	//Alarm Priority setpoint
	{attribute 'OPC.UA.DA' :='1'}
	popa_0081_lt_3202_a_high_high_priority : INT;
	//Alarm delay setpoint(seconds)
	{attribute 'OPC.UA.DA' :='1'}
	popa_0081_lt_3202_a_high_high_delay_setpoint : INT;
	//Alarm active for HMI
	{attribute 'OPC.UA.DA' :='1'}
	popa_0081_lt_3202_a_high_high_active : BOOL;
	//Analog Alarm Setpoint
	{attribute 'OPC.UA.DA' :='1'}
	popa_0081_lt_3202_a_high_high_setpoint : REAL;
	//Alarm enable
	{attribute 'OPC.UA.DA' :='1'}
	popa_0081_lt_3202_a_high_high_enable: BOOL;
	
	
	//Raw Min value for analog input
	{attribute 'OPC.UA.DA' :='1'}
	popa_0081_lt_3202_a_raw_min : REAL :=0;
	//Raw max value for analog input
	{attribute 'OPC.UA.DA' :='1'}
	popa_0081_lt_3202_a_raw_max : REAL :=32767;
	//EU Min value for analog input
	{attribute 'OPC.UA.DA' :='1'}
	popa_0081_lt_3202_a_eu_min : REAL;
	//EU Max value for analog input
	{attribute 'OPC.UA.DA' :='1'}
	popa_0081_lt_3202_a_eu_max : REAL;
	//Filter factor value for analog input
	{attribute 'OPC.UA.DA' :='1'}
	popa_0081_lt_3202_a_filter_factor : REAL;
	//Scaled value for analog input
	{attribute 'OPC.UA.DA' :='1'}
	popa_0081_lt_3202_a_scaled_value : REAL;
	
	//---lt_3302-----------------------------------------------------------------------------------------------------------------------
	//Alarm Priority setpoint
	{attribute 'OPC.UA.DA' :='1'}
	popa_0081_lt_3302_a_low_low_priority : INT;
	//Alarm delay setpoint(seconds)
	{attribute 'OPC.UA.DA' :='1'}
	popa_0081_lt_3302_a_low_low_delay_setpoint : INT;
	//Alarm active for HMI
	{attribute 'OPC.UA.DA' :='1'}
	popa_0081_lt_3302_a_low_low_active : BOOL;
	//Analog Alarm Setpoint
	{attribute 'OPC.UA.DA' :='1'}
	popa_0081_lt_3302_a_low_low_setpoint : REAL;
	//Alarm enable
	{attribute 'OPC.UA.DA' :='1'}
	popa_0081_lt_3302_a_low_low_enable: BOOL;
	
	//Alarm Priority setpoint
	{attribute 'OPC.UA.DA' :='1'}
	popa_0081_lt_3302_a_low_priority : INT;
	//Alarm delay setpoint(seconds)
	{attribute 'OPC.UA.DA' :='1'}
	popa_0081_lt_3302_a_low_delay_setpoint : INT;
	//Alarm active for HMI
	{attribute 'OPC.UA.DA' :='1'}
	popa_0081_lt_3302_a_low_active : BOOL;
	//Analog Alarm Setpoint
	{attribute 'OPC.UA.DA' :='1'}
	popa_0081_lt_3302_a_low_setpoint : REAL;
	//Alarm enable
	{attribute 'OPC.UA.DA' :='1'}
	popa_0081_lt_3302_a_low_enable: BOOL;
	
	//Alarm Priority setpoint
	{attribute 'OPC.UA.DA' :='1'}
	popa_0081_lt_3302_a_high_priority : INT;
	//Alarm delay setpoint(seconds)
	{attribute 'OPC.UA.DA' :='1'}
	popa_0081_lt_3302_a_high_delay_setpoint : INT;
	//Alarm active for HMI
	{attribute 'OPC.UA.DA' :='1'}
	popa_0081_lt_3302_a_high_active : BOOL;
	//Analog Alarm Setpoint
	{attribute 'OPC.UA.DA' :='1'}
	popa_0081_lt_3302_a_high_setpoint : REAL;
	//Alarm enable
	{attribute 'OPC.UA.DA' :='1'}
	popa_0081_lt_3302_a_high_enable: BOOL;
	
	//Alarm Priority setpoint
	{attribute 'OPC.UA.DA' :='1'}
	popa_0081_lt_3302_a_high_high_priority : INT;
	//Alarm delay setpoint(seconds)
	{attribute 'OPC.UA.DA' :='1'}
	popa_0081_lt_3302_a_high_high_delay_setpoint : INT;
	//Alarm active for HMI
	{attribute 'OPC.UA.DA' :='1'}
	popa_0081_lt_3302_a_high_high_active : BOOL;
	//Analog Alarm Setpoint
	{attribute 'OPC.UA.DA' :='1'}
	popa_0081_lt_3302_a_high_high_setpoint : REAL;
	//Alarm enable
	{attribute 'OPC.UA.DA' :='1'}
	popa_0081_lt_3302_a_high_high_enable: BOOL;
	
	
	//Raw Min value for analog input
	{attribute 'OPC.UA.DA' :='1'}
	popa_0081_lt_3302_a_raw_min : REAL :=0;
	//Raw max value for analog input
	{attribute 'OPC.UA.DA' :='1'}
	popa_0081_lt_3302_a_raw_max : REAL :=32767;
	//EU Min value for analog input
	{attribute 'OPC.UA.DA' :='1'}
	popa_0081_lt_3302_a_eu_min : REAL;
	//EU Max value for analog input
	{attribute 'OPC.UA.DA' :='1'}
	popa_0081_lt_3302_a_eu_max : REAL;
	//Filter factor value for analog input
	{attribute 'OPC.UA.DA' :='1'}
	popa_0081_lt_3302_a_filter_factor : REAL;
	//Scaled value for analog input
	{attribute 'OPC.UA.DA' :='1'}
	popa_0081_lt_3302_a_scaled_value : REAL;
	
	//---lt_3153-----------------------------------------------------------------------------------------------------------------------
	//Alarm Priority setpoint
	{attribute 'OPC.UA.DA' :='1'}
	popa_0081_lt_3153_a_low_low_priority : INT;
	//Alarm delay setpoint(seconds)
	{attribute 'OPC.UA.DA' :='1'}
	popa_0081_lt_3153_a_low_low_delay_setpoint : INT;
	//Alarm active for HMI
	{attribute 'OPC.UA.DA' :='1'}
	popa_0081_lt_3153_a_low_low_active : BOOL;
	//Analog Alarm Setpoint
	{attribute 'OPC.UA.DA' :='1'}
	popa_0081_lt_3153_a_low_low_setpoint : REAL;
	//Alarm enable
	{attribute 'OPC.UA.DA' :='1'}
	popa_0081_lt_3153_a_low_low_enable: BOOL;
	
	//Alarm Priority setpoint
	{attribute 'OPC.UA.DA' :='1'}
	popa_0081_lt_3153_a_low_priority : INT;
	//Alarm delay setpoint(seconds)
	{attribute 'OPC.UA.DA' :='1'}
	popa_0081_lt_3153_a_low_delay_setpoint : INT;
	//Alarm active for HMI
	{attribute 'OPC.UA.DA' :='1'}
	popa_0081_lt_3153_a_low_active : BOOL;
	//Analog Alarm Setpoint
	{attribute 'OPC.UA.DA' :='1'}
	popa_0081_lt_3153_a_low_setpoint : REAL;
	//Alarm enable
	{attribute 'OPC.UA.DA' :='1'}
	popa_0081_lt_3153_a_low_enable: BOOL;
	
	//Alarm Priority setpoint
	{attribute 'OPC.UA.DA' :='1'}
	popa_0081_lt_3153_a_high_priority : INT;
	//Alarm delay setpoint(seconds)
	{attribute 'OPC.UA.DA' :='1'}
	popa_0081_lt_3153_a_high_delay_setpoint : INT;
	//Alarm active for HMI
	{attribute 'OPC.UA.DA' :='1'}
	popa_0081_lt_3153_a_high_active : BOOL;
	//Analog Alarm Setpoint
	{attribute 'OPC.UA.DA' :='1'}
	popa_0081_lt_3153_a_high_setpoint : REAL;
	//Alarm enable
	{attribute 'OPC.UA.DA' :='1'}
	popa_0081_lt_3153_a_high_enable: BOOL;
	
	//Alarm Priority setpoint
	{attribute 'OPC.UA.DA' :='1'}
	popa_0081_lt_3153_a_high_high_priority : INT;
	//Alarm delay setpoint(seconds)
	{attribute 'OPC.UA.DA' :='1'}
	popa_0081_lt_3153_a_high_high_delay_setpoint : INT;
	//Alarm active for HMI
	{attribute 'OPC.UA.DA' :='1'}
	popa_0081_lt_3153_a_high_high_active : BOOL;
	//Analog Alarm Setpoint
	{attribute 'OPC.UA.DA' :='1'}
	popa_0081_lt_3153_a_high_high_setpoint : REAL;
	//Alarm enable
	{attribute 'OPC.UA.DA' :='1'}
	popa_0081_lt_3153_a_high_high_enable: BOOL;
	
	
	//Raw Min value for analog input
	{attribute 'OPC.UA.DA' :='1'}
	popa_0081_lt_3153_a_raw_min : REAL :=0;
	//Raw max value for analog input
	{attribute 'OPC.UA.DA' :='1'}
	popa_0081_lt_3153_a_raw_max : REAL :=32767;
	//EU Min value for analog input
	{attribute 'OPC.UA.DA' :='1'}
	popa_0081_lt_3153_a_eu_min : REAL;
	//EU Max value for analog input
	{attribute 'OPC.UA.DA' :='1'}
	popa_0081_lt_3153_a_eu_max : REAL;
	//Filter factor value for analog input
	{attribute 'OPC.UA.DA' :='1'}
	popa_0081_lt_3153_a_filter_factor : REAL;
	//Scaled value for analog input
	{attribute 'OPC.UA.DA' :='1'}
	popa_0081_lt_3153_a_scaled_value : REAL;
	
	//---lt_3253-----------------------------------------------------------------------------------------------------------------------
	//Alarm Priority setpoint
	{attribute 'OPC.UA.DA' :='1'}
	popa_0081_lt_3253_a_low_low_priority : INT;
	//Alarm delay setpoint(seconds)
	{attribute 'OPC.UA.DA' :='1'}
	popa_0081_lt_3253_a_low_low_delay_setpoint : INT;
	//Alarm active for HMI
	{attribute 'OPC.UA.DA' :='1'}
	popa_0081_lt_3253_a_low_low_active : BOOL;
	//Analog Alarm Setpoint
	{attribute 'OPC.UA.DA' :='1'}
	popa_0081_lt_3253_a_low_low_setpoint : REAL;
	//Alarm enable
	{attribute 'OPC.UA.DA' :='1'}
	popa_0081_lt_3253_a_low_low_enable: BOOL;
	
	//Alarm Priority setpoint
	{attribute 'OPC.UA.DA' :='1'}
	popa_0081_lt_3253_a_low_priority : INT;
	//Alarm delay setpoint(seconds)
	{attribute 'OPC.UA.DA' :='1'}
	popa_0081_lt_3253_a_low_delay_setpoint : INT;
	//Alarm active for HMI
	{attribute 'OPC.UA.DA' :='1'}
	popa_0081_lt_3253_a_low_active : BOOL;
	//Analog Alarm Setpoint
	{attribute 'OPC.UA.DA' :='1'}
	popa_0081_lt_3253_a_low_setpoint : REAL;
	//Alarm enable
	{attribute 'OPC.UA.DA' :='1'}
	popa_0081_lt_3253_a_low_enable: BOOL;
	
	//Alarm Priority setpoint
	{attribute 'OPC.UA.DA' :='1'}
	popa_0081_lt_3253_a_high_priority : INT;
	//Alarm delay setpoint(seconds)
	{attribute 'OPC.UA.DA' :='1'}
	popa_0081_lt_3253_a_high_delay_setpoint : INT;
	//Alarm active for HMI
	{attribute 'OPC.UA.DA' :='1'}
	popa_0081_lt_3253_a_high_active : BOOL;
	//Analog Alarm Setpoint
	{attribute 'OPC.UA.DA' :='1'}
	popa_0081_lt_3253_a_high_setpoint : REAL;
	//Alarm enable
	{attribute 'OPC.UA.DA' :='1'}
	popa_0081_lt_3253_a_high_enable: BOOL;
	
	//Alarm Priority setpoint
	{attribute 'OPC.UA.DA' :='1'}
	popa_0081_lt_3253_a_high_high_priority : INT;
	//Alarm delay setpoint(seconds)
	{attribute 'OPC.UA.DA' :='1'}
	popa_0081_lt_3253_a_high_high_delay_setpoint : INT;
	//Alarm active for HMI
	{attribute 'OPC.UA.DA' :='1'}
	popa_0081_lt_3253_a_high_high_active : BOOL;
	//Analog Alarm Setpoint
	{attribute 'OPC.UA.DA' :='1'}
	popa_0081_lt_3253_a_high_high_setpoint : REAL;
	//Alarm enable
	{attribute 'OPC.UA.DA' :='1'}
	popa_0081_lt_3253_a_high_high_enable: BOOL;
	
	
	//Raw Min value for analog input
	{attribute 'OPC.UA.DA' :='1'}
	popa_0081_lt_3253_a_raw_min : REAL :=0;
	//Raw max value for analog input
	{attribute 'OPC.UA.DA' :='1'}
	popa_0081_lt_3253_a_raw_max : REAL :=32767;
	//EU Min value for analog input
	{attribute 'OPC.UA.DA' :='1'}
	popa_0081_lt_3253_a_eu_min : REAL;
	//EU Max value for analog input
	{attribute 'OPC.UA.DA' :='1'}
	popa_0081_lt_3253_a_eu_max : REAL;
	//Filter factor value for analog input
	{attribute 'OPC.UA.DA' :='1'}
	popa_0081_lt_3253_a_filter_factor : REAL;
	//Scaled value for analog input
	{attribute 'OPC.UA.DA' :='1'}
	popa_0081_lt_3253_a_scaled_value : REAL;
	
	//---lt_3353-----------------------------------------------------------------------------------------------------------------------
	//Alarm Priority setpoint
	{attribute 'OPC.UA.DA' :='1'}
	popa_0081_lt_3353_a_low_low_priority : INT;
	//Alarm delay setpoint(seconds)
	{attribute 'OPC.UA.DA' :='1'}
	popa_0081_lt_3353_a_low_low_delay_setpoint : INT;
	//Alarm active for HMI
	{attribute 'OPC.UA.DA' :='1'}
	popa_0081_lt_3353_a_low_low_active : BOOL;
	//Analog Alarm Setpoint
	{attribute 'OPC.UA.DA' :='1'}
	popa_0081_lt_3353_a_low_low_setpoint : REAL;
	//Alarm enable
	{attribute 'OPC.UA.DA' :='1'}
	popa_0081_lt_3353_a_low_low_enable: BOOL;
	
	//Alarm Priority setpoint
	{attribute 'OPC.UA.DA' :='1'}
	popa_0081_lt_3353_a_low_priority : INT;
	//Alarm delay setpoint(seconds)
	{attribute 'OPC.UA.DA' :='1'}
	popa_0081_lt_3353_a_low_delay_setpoint : INT;
	//Alarm active for HMI
	{attribute 'OPC.UA.DA' :='1'}
	popa_0081_lt_3353_a_low_active : BOOL;
	//Analog Alarm Setpoint
	{attribute 'OPC.UA.DA' :='1'}
	popa_0081_lt_3353_a_low_setpoint : REAL;
	//Alarm enable
	{attribute 'OPC.UA.DA' :='1'}
	popa_0081_lt_3353_a_low_enable: BOOL;
	
	//Alarm Priority setpoint
	{attribute 'OPC.UA.DA' :='1'}
	popa_0081_lt_3353_a_high_priority : INT;
	//Alarm delay setpoint(seconds)
	{attribute 'OPC.UA.DA' :='1'}
	popa_0081_lt_3353_a_high_delay_setpoint : INT;
	//Alarm active for HMI
	{attribute 'OPC.UA.DA' :='1'}
	popa_0081_lt_3353_a_high_active : BOOL;
	//Analog Alarm Setpoint
	{attribute 'OPC.UA.DA' :='1'}
	popa_0081_lt_3353_a_high_setpoint : REAL;
	//Alarm enable
	{attribute 'OPC.UA.DA' :='1'}
	popa_0081_lt_3353_a_high_enable: BOOL;
	
	//Alarm Priority setpoint
	{attribute 'OPC.UA.DA' :='1'}
	popa_0081_lt_3353_a_high_high_priority : INT;
	//Alarm delay setpoint(seconds)
	{attribute 'OPC.UA.DA' :='1'}
	popa_0081_lt_3353_a_high_high_delay_setpoint : INT;
	//Alarm active for HMI
	{attribute 'OPC.UA.DA' :='1'}
	popa_0081_lt_3353_a_high_high_active : BOOL;
	//Analog Alarm Setpoint
	{attribute 'OPC.UA.DA' :='1'}
	popa_0081_lt_3353_a_high_high_setpoint : REAL;
	//Alarm enable
	{attribute 'OPC.UA.DA' :='1'}
	popa_0081_lt_3353_a_high_high_enable: BOOL;
	
	
	//Raw Min value for analog input
	{attribute 'OPC.UA.DA' :='1'}
	popa_0081_lt_3353_a_raw_min : REAL :=0;
	//Raw max value for analog input
	{attribute 'OPC.UA.DA' :='1'}
	popa_0081_lt_3353_a_raw_max : REAL :=32767;
	//EU Min value for analog input
	{attribute 'OPC.UA.DA' :='1'}
	popa_0081_lt_3353_a_eu_min : REAL;
	//EU Max value for analog input
	{attribute 'OPC.UA.DA' :='1'}
	popa_0081_lt_3353_a_eu_max : REAL;
	//Filter factor value for analog input
	{attribute 'OPC.UA.DA' :='1'}
	popa_0081_lt_3353_a_filter_factor : REAL;
	//Scaled value for analog input
	{attribute 'OPC.UA.DA' :='1'}
	popa_0081_lt_3353_a_scaled_value : REAL;
	
	//---lt_3402-----------------------------------------------------------------------------------------------------------------------
	//Alarm Priority setpoint
	{attribute 'OPC.UA.DA' :='1'}
	popa_0091_lt_3402_a_low_low_priority : INT;
	//Alarm delay setpoint(seconds)
	{attribute 'OPC.UA.DA' :='1'}
	popa_0091_lt_3402_a_low_low_delay_setpoint : INT;
	//Alarm active for HMI
	{attribute 'OPC.UA.DA' :='1'}
	popa_0091_lt_3402_a_low_low_active : BOOL;
	//Analog Alarm Setpoint
	{attribute 'OPC.UA.DA' :='1'}
	popa_0091_lt_3402_a_low_low_setpoint : REAL;
	//Alarm enable
	{attribute 'OPC.UA.DA' :='1'}
	popa_0091_lt_3402_a_low_low_enable: BOOL;
	
	//Alarm Priority setpoint
	{attribute 'OPC.UA.DA' :='1'}
	popa_0091_lt_3402_a_low_priority : INT;
	//Alarm delay setpoint(seconds)
	{attribute 'OPC.UA.DA' :='1'}
	popa_0091_lt_3402_a_low_delay_setpoint : INT;
	//Alarm active for HMI
	{attribute 'OPC.UA.DA' :='1'}
	popa_0091_lt_3402_a_low_active : BOOL;
	//Analog Alarm Setpoint
	{attribute 'OPC.UA.DA' :='1'}
	popa_0091_lt_3402_a_low_setpoint : REAL;
	//Alarm enable
	{attribute 'OPC.UA.DA' :='1'}
	popa_0091_lt_3402_a_low_enable: BOOL;
	
	//Alarm Priority setpoint
	{attribute 'OPC.UA.DA' :='1'}
	popa_0091_lt_3402_a_high_priority : INT;
	//Alarm delay setpoint(seconds)
	{attribute 'OPC.UA.DA' :='1'}
	popa_0091_lt_3402_a_high_delay_setpoint : INT;
	//Alarm active for HMI
	{attribute 'OPC.UA.DA' :='1'}
	popa_0091_lt_3402_a_high_active : BOOL;
	//Analog Alarm Setpoint
	{attribute 'OPC.UA.DA' :='1'}
	popa_0091_lt_3402_a_high_setpoint : REAL;
	//Alarm enable
	{attribute 'OPC.UA.DA' :='1'}
	popa_0091_lt_3402_a_high_enable: BOOL;
	
	//Alarm Priority setpoint
	{attribute 'OPC.UA.DA' :='1'}
	popa_0091_lt_3402_a_high_high_priority : INT;
	//Alarm delay setpoint(seconds)
	{attribute 'OPC.UA.DA' :='1'}
	popa_0091_lt_3402_a_high_high_delay_setpoint : INT;
	//Alarm active for HMI
	{attribute 'OPC.UA.DA' :='1'}
	popa_0091_lt_3402_a_high_high_active : BOOL;
	//Analog Alarm Setpoint
	{attribute 'OPC.UA.DA' :='1'}
	popa_0091_lt_3402_a_high_high_setpoint : REAL;
	//Alarm enable
	{attribute 'OPC.UA.DA' :='1'}
	popa_0091_lt_3402_a_high_high_enable: BOOL;
	
	
	//Raw Min value for analog input
	{attribute 'OPC.UA.DA' :='1'}
	popa_0091_lt_3402_a_raw_min : REAL :=0;
	//Raw max value for analog input
	{attribute 'OPC.UA.DA' :='1'}
	popa_0091_lt_3402_a_raw_max : REAL :=32767;
	//EU Min value for analog input
	{attribute 'OPC.UA.DA' :='1'}
	popa_0091_lt_3402_a_eu_min : REAL;
	//EU Max value for analog input
	{attribute 'OPC.UA.DA' :='1'}
	popa_0091_lt_3402_a_eu_max : REAL;
	//Filter factor value for analog input
	{attribute 'OPC.UA.DA' :='1'}
	popa_0091_lt_3402_a_filter_factor : REAL;
	//Scaled value for analog input
	{attribute 'OPC.UA.DA' :='1'}
	popa_0091_lt_3402_a_scaled_value : REAL;
	
	
	//---pt_3119-----------------------------------------------------------------------------------------------------------------------
	//Alarm Priority setpoint
	{attribute 'OPC.UA.DA' :='1'}
	popa_0081_pt_3119_a_low_low_priority : INT;
	//Alarm delay setpoint(seconds)
	{attribute 'OPC.UA.DA' :='1'}
	popa_0081_pt_3119_a_low_low_delay_setpoint : INT;
	//Alarm active for HMI
	{attribute 'OPC.UA.DA' :='1'}
	popa_0081_pt_3119_a_low_low_active : BOOL;
	//Analog Alarm Setpoint
	{attribute 'OPC.UA.DA' :='1'}
	popa_0081_pt_3119_a_low_low_setpoint : REAL;
	//Alarm enable
	{attribute 'OPC.UA.DA' :='1'}
	popa_0081_pt_3119_a_low_low_enable: BOOL;
	
	//Alarm Priority setpoint
	{attribute 'OPC.UA.DA' :='1'}
	popa_0081_pt_3119_a_low_priority : INT;
	//Alarm delay setpoint(seconds)
	{attribute 'OPC.UA.DA' :='1'}
	popa_0081_pt_3119_a_low_delay_setpoint : INT;
	//Alarm active for HMI
	{attribute 'OPC.UA.DA' :='1'}
	popa_0081_pt_3119_a_low_active : BOOL;
	//Analog Alarm Setpoint
	{attribute 'OPC.UA.DA' :='1'}
	popa_0081_pt_3119_a_low_setpoint : REAL;
	//Alarm enable
	{attribute 'OPC.UA.DA' :='1'}
	popa_0081_pt_3119_a_low_enable: BOOL;
	
	//Alarm Priority setpoint
	{attribute 'OPC.UA.DA' :='1'}
	popa_0081_pt_3119_a_high_priority : INT;
	//Alarm delay setpoint(seconds)
	{attribute 'OPC.UA.DA' :='1'}
	popa_0081_pt_3119_a_high_delay_setpoint : INT;
	//Alarm active for HMI
	{attribute 'OPC.UA.DA' :='1'}
	popa_0081_pt_3119_a_high_active : BOOL;
	//Analog Alarm Setpoint
	{attribute 'OPC.UA.DA' :='1'}
	popa_0081_pt_3119_a_high_setpoint : REAL;
	//Alarm enable
	{attribute 'OPC.UA.DA' :='1'}
	popa_0081_pt_3119_a_high_enable: BOOL;
	
	//Alarm Priority setpoint
	{attribute 'OPC.UA.DA' :='1'}
	popa_0081_pt_3119_a_high_high_priority : INT;
	//Alarm delay setpoint(seconds)
	{attribute 'OPC.UA.DA' :='1'}
	popa_0081_pt_3119_a_high_high_delay_setpoint : INT;
	//Alarm active for HMI
	{attribute 'OPC.UA.DA' :='1'}
	popa_0081_pt_3119_a_high_high_active : BOOL;
	//Analog Alarm Setpoint
	{attribute 'OPC.UA.DA' :='1'}
	popa_0081_pt_3119_a_high_high_setpoint : REAL;
	//Alarm enable
	{attribute 'OPC.UA.DA' :='1'}
	popa_0081_pt_3119_a_high_high_enable: BOOL;
	
	
	//Raw Min value for analog input
	{attribute 'OPC.UA.DA' :='1'}
	popa_0081_pt_3119_a_raw_min : REAL :=0;
	//Raw max value for analog input
	{attribute 'OPC.UA.DA' :='1'}
	popa_0081_pt_3119_a_raw_max : REAL :=32767;
	//EU Min value for analog input
	{attribute 'OPC.UA.DA' :='1'}
	popa_0081_pt_3119_a_eu_min : REAL;
	//EU Max value for analog input
	{attribute 'OPC.UA.DA' :='1'}
	popa_0081_pt_3119_a_eu_max : REAL;
	//Filter factor value for analog input
	{attribute 'OPC.UA.DA' :='1'}
	popa_0081_pt_3119_a_filter_factor : REAL;
	//Scaled value for analog input
	{attribute 'OPC.UA.DA' :='1'}
	popa_0081_pt_3119_a_scaled_value : REAL;
	
	//---pt_3219-----------------------------------------------------------------------------------------------------------------------
	//Alarm Priority setpoint
	{attribute 'OPC.UA.DA' :='1'}
	popa_0081_pt_3219_a_low_low_priority : INT;
	//Alarm delay setpoint(seconds)
	{attribute 'OPC.UA.DA' :='1'}
	popa_0081_pt_3219_a_low_low_delay_setpoint : INT;
	//Alarm active for HMI
	{attribute 'OPC.UA.DA' :='1'}
	popa_0081_pt_3219_a_low_low_active : BOOL;
	//Analog Alarm Setpoint
	{attribute 'OPC.UA.DA' :='1'}
	popa_0081_pt_3219_a_low_low_setpoint : REAL;
	//Alarm enable
	{attribute 'OPC.UA.DA' :='1'}
	popa_0081_pt_3219_a_low_low_enable: BOOL;
	
	//Alarm Priority setpoint
	{attribute 'OPC.UA.DA' :='1'}
	popa_0081_pt_3219_a_low_priority : INT;
	//Alarm delay setpoint(seconds)
	{attribute 'OPC.UA.DA' :='1'}
	popa_0081_pt_3219_a_low_delay_setpoint : INT;
	//Alarm active for HMI
	{attribute 'OPC.UA.DA' :='1'}
	popa_0081_pt_3219_a_low_active : BOOL;
	//Analog Alarm Setpoint
	{attribute 'OPC.UA.DA' :='1'}
	popa_0081_pt_3219_a_low_setpoint : REAL;
	//Alarm enable
	{attribute 'OPC.UA.DA' :='1'}
	popa_0081_pt_3219_a_low_enable: BOOL;
	
	//Alarm Priority setpoint
	{attribute 'OPC.UA.DA' :='1'}
	popa_0081_pt_3219_a_high_priority : INT;
	//Alarm delay setpoint(seconds)
	{attribute 'OPC.UA.DA' :='1'}
	popa_0081_pt_3219_a_high_delay_setpoint : INT;
	//Alarm active for HMI
	{attribute 'OPC.UA.DA' :='1'}
	popa_0081_pt_3219_a_high_active : BOOL;
	//Analog Alarm Setpoint
	{attribute 'OPC.UA.DA' :='1'}
	popa_0081_pt_3219_a_high_setpoint : REAL;
	//Alarm enable
	{attribute 'OPC.UA.DA' :='1'}
	popa_0081_pt_3219_a_high_enable: BOOL;
	
	//Alarm Priority setpoint
	{attribute 'OPC.UA.DA' :='1'}
	popa_0081_pt_3219_a_high_high_priority : INT;
	//Alarm delay setpoint(seconds)
	{attribute 'OPC.UA.DA' :='1'}
	popa_0081_pt_3219_a_high_high_delay_setpoint : INT;
	//Alarm active for HMI
	{attribute 'OPC.UA.DA' :='1'}
	popa_0081_pt_3219_a_high_high_active : BOOL;
	//Analog Alarm Setpoint
	{attribute 'OPC.UA.DA' :='1'}
	popa_0081_pt_3219_a_high_high_setpoint : REAL;
	//Alarm enable
	{attribute 'OPC.UA.DA' :='1'}
	popa_0081_pt_3219_a_high_high_enable: BOOL;
	
	
	//Raw Min value for analog input
	{attribute 'OPC.UA.DA' :='1'}
	popa_0081_pt_3219_a_raw_min : REAL :=0;
	//Raw max value for analog input
	{attribute 'OPC.UA.DA' :='1'}
	popa_0081_pt_3219_a_raw_max : REAL :=32767;
	//EU Min value for analog input
	{attribute 'OPC.UA.DA' :='1'}
	popa_0081_pt_3219_a_eu_min : REAL;
	//EU Max value for analog input
	{attribute 'OPC.UA.DA' :='1'}
	popa_0081_pt_3219_a_eu_max : REAL;
	//Filter factor value for analog input
	{attribute 'OPC.UA.DA' :='1'}
	popa_0081_pt_3219_a_filter_factor : REAL;
	//Scaled value for analog input
	{attribute 'OPC.UA.DA' :='1'}
	popa_0081_pt_3219_a_scaled_value : REAL;
	
	//---pt_3319-----------------------------------------------------------------------------------------------------------------------
	//Alarm Priority setpoint
	{attribute 'OPC.UA.DA' :='1'}
	popa_0081_pt_3319_a_low_low_priority : INT;
	//Alarm delay setpoint(seconds)
	{attribute 'OPC.UA.DA' :='1'}
	popa_0081_pt_3319_a_low_low_delay_setpoint : INT;
	//Alarm active for HMI
	{attribute 'OPC.UA.DA' :='1'}
	popa_0081_pt_3319_a_low_low_active : BOOL;
	//Analog Alarm Setpoint
	{attribute 'OPC.UA.DA' :='1'}
	popa_0081_pt_3319_a_low_low_setpoint : REAL;
	//Alarm enable
	{attribute 'OPC.UA.DA' :='1'}
	popa_0081_pt_3319_a_low_low_enable: BOOL;
	
	//Alarm Priority setpoint
	{attribute 'OPC.UA.DA' :='1'}
	popa_0081_pt_3319_a_low_priority : INT;
	//Alarm delay setpoint(seconds)
	{attribute 'OPC.UA.DA' :='1'}
	popa_0081_pt_3319_a_low_delay_setpoint : INT;
	//Alarm active for HMI
	{attribute 'OPC.UA.DA' :='1'}
	popa_0081_pt_3319_a_low_active : BOOL;
	//Analog Alarm Setpoint
	{attribute 'OPC.UA.DA' :='1'}
	popa_0081_pt_3319_a_low_setpoint : REAL;
	//Alarm enable
	{attribute 'OPC.UA.DA' :='1'}
	popa_0081_pt_3319_a_low_enable: BOOL;
	
	//Alarm Priority setpoint
	{attribute 'OPC.UA.DA' :='1'}
	popa_0081_pt_3319_a_high_priority : INT;
	//Alarm delay setpoint(seconds)
	{attribute 'OPC.UA.DA' :='1'}
	popa_0081_pt_3319_a_high_delay_setpoint : INT;
	//Alarm active for HMI
	{attribute 'OPC.UA.DA' :='1'}
	popa_0081_pt_3319_a_high_active : BOOL;
	//Analog Alarm Setpoint
	{attribute 'OPC.UA.DA' :='1'}
	popa_0081_pt_3319_a_high_setpoint : REAL;
	//Alarm enable
	{attribute 'OPC.UA.DA' :='1'}
	popa_0081_pt_3319_a_high_enable: BOOL;
	
	//Alarm Priority setpoint
	{attribute 'OPC.UA.DA' :='1'}
	popa_0081_pt_3319_a_high_high_priority : INT;
	//Alarm delay setpoint(seconds)
	{attribute 'OPC.UA.DA' :='1'}
	popa_0081_pt_3319_a_high_high_delay_setpoint : INT;
	//Alarm active for HMI
	{attribute 'OPC.UA.DA' :='1'}
	popa_0081_pt_3319_a_high_high_active : BOOL;
	//Analog Alarm Setpoint
	{attribute 'OPC.UA.DA' :='1'}
	popa_0081_pt_3319_a_high_high_setpoint : REAL;
	//Alarm enable
	{attribute 'OPC.UA.DA' :='1'}
	popa_0081_pt_3319_a_high_high_enable: BOOL;
	
	
	//Raw Min value for analog input
	{attribute 'OPC.UA.DA' :='1'}
	popa_0081_pt_3319_a_raw_min : REAL :=0;
	//Raw max value for analog input
	{attribute 'OPC.UA.DA' :='1'}
	popa_0081_pt_3319_a_raw_max : REAL :=32767;
	//EU Min value for analog input
	{attribute 'OPC.UA.DA' :='1'}
	popa_0081_pt_3319_a_eu_min : REAL;
	//EU Max value for analog input
	{attribute 'OPC.UA.DA' :='1'}
	popa_0081_pt_3319_a_eu_max : REAL;
	//Filter factor value for analog input
	{attribute 'OPC.UA.DA' :='1'}
	popa_0081_pt_3319_a_filter_factor : REAL;
	//Scaled value for analog input
	{attribute 'OPC.UA.DA' :='1'}
	popa_0081_pt_3319_a_scaled_value : REAL;
	
	//---pt_3141-----------------------------------------------------------------------------------------------------------------------
	//Alarm Priority setpoint
	{attribute 'OPC.UA.DA' :='1'}
	popa_0081_pt_3141_a_low_low_priority : INT;
	//Alarm delay setpoint(seconds)
	{attribute 'OPC.UA.DA' :='1'}
	popa_0081_pt_3141_a_low_low_delay_setpoint : INT;
	//Alarm active for HMI
	{attribute 'OPC.UA.DA' :='1'}
	popa_0081_pt_3141_a_low_low_active : BOOL;
	//Analog Alarm Setpoint
	{attribute 'OPC.UA.DA' :='1'}
	popa_0081_pt_3141_a_low_low_setpoint : REAL;
	//Alarm enable
	{attribute 'OPC.UA.DA' :='1'}
	popa_0081_pt_3141_a_low_low_enable: BOOL;
	
	//Alarm Priority setpoint
	{attribute 'OPC.UA.DA' :='1'}
	popa_0081_pt_3141_a_low_priority : INT;
	//Alarm delay setpoint(seconds)
	{attribute 'OPC.UA.DA' :='1'}
	popa_0081_pt_3141_a_low_delay_setpoint : INT;
	//Alarm active for HMI
	{attribute 'OPC.UA.DA' :='1'}
	popa_0081_pt_3141_a_low_active : BOOL;
	//Analog Alarm Setpoint
	{attribute 'OPC.UA.DA' :='1'}
	popa_0081_pt_3141_a_low_setpoint : REAL;
	//Alarm enable
	{attribute 'OPC.UA.DA' :='1'}
	popa_0081_pt_3141_a_low_enable: BOOL;
	
	//Alarm Priority setpoint
	{attribute 'OPC.UA.DA' :='1'}
	popa_0081_pt_3141_a_high_priority : INT;
	//Alarm delay setpoint(seconds)
	{attribute 'OPC.UA.DA' :='1'}
	popa_0081_pt_3141_a_high_delay_setpoint : INT;
	//Alarm active for HMI
	{attribute 'OPC.UA.DA' :='1'}
	popa_0081_pt_3141_a_high_active : BOOL;
	//Analog Alarm Setpoint
	{attribute 'OPC.UA.DA' :='1'}
	popa_0081_pt_3141_a_high_setpoint : REAL;
	//Alarm enable
	{attribute 'OPC.UA.DA' :='1'}
	popa_0081_pt_3141_a_high_enable: BOOL;
	
	//Alarm Priority setpoint
	{attribute 'OPC.UA.DA' :='1'}
	popa_0081_pt_3141_a_high_high_priority : INT;
	//Alarm delay setpoint(seconds)
	{attribute 'OPC.UA.DA' :='1'}
	popa_0081_pt_3141_a_high_high_delay_setpoint : INT;
	//Alarm active for HMI
	{attribute 'OPC.UA.DA' :='1'}
	popa_0081_pt_3141_a_high_high_active : BOOL;
	//Analog Alarm Setpoint
	{attribute 'OPC.UA.DA' :='1'}
	popa_0081_pt_3141_a_high_high_setpoint : REAL;
	//Alarm enable
	{attribute 'OPC.UA.DA' :='1'}
	popa_0081_pt_3141_a_high_high_enable: BOOL;
	
	
	//Raw Min value for analog input
	{attribute 'OPC.UA.DA' :='1'}
	popa_0081_pt_3141_a_raw_min : REAL :=0;
	//Raw max value for analog input
	{attribute 'OPC.UA.DA' :='1'}
	popa_0081_pt_3141_a_raw_max : REAL :=32767;
	//EU Min value for analog input
	{attribute 'OPC.UA.DA' :='1'}
	popa_0081_pt_3141_a_eu_min : REAL;
	//EU Max value for analog input
	{attribute 'OPC.UA.DA' :='1'}
	popa_0081_pt_3141_a_eu_max : REAL;
	//Filter factor value for analog input
	{attribute 'OPC.UA.DA' :='1'}
	popa_0081_pt_3141_a_filter_factor : REAL;
	//Scaled value for analog input
	{attribute 'OPC.UA.DA' :='1'}
	popa_0081_pt_3141_a_scaled_value : REAL;
	
	//---pt_3241-----------------------------------------------------------------------------------------------------------------------
	//Alarm Priority setpoint
	{attribute 'OPC.UA.DA' :='1'}
	popa_0081_pt_3241_a_low_low_priority : INT;
	//Alarm delay setpoint(seconds)
	{attribute 'OPC.UA.DA' :='1'}
	popa_0081_pt_3241_a_low_low_delay_setpoint : INT;
	//Alarm active for HMI
	{attribute 'OPC.UA.DA' :='1'}
	popa_0081_pt_3241_a_low_low_active : BOOL;
	//Analog Alarm Setpoint
	{attribute 'OPC.UA.DA' :='1'}
	popa_0081_pt_3241_a_low_low_setpoint : REAL;
	//Alarm enable
	{attribute 'OPC.UA.DA' :='1'}
	popa_0081_pt_3241_a_low_low_enable: BOOL;
	
	//Alarm Priority setpoint
	{attribute 'OPC.UA.DA' :='1'}
	popa_0081_pt_3241_a_low_priority : INT;
	//Alarm delay setpoint(seconds)
	{attribute 'OPC.UA.DA' :='1'}
	popa_0081_pt_3241_a_low_delay_setpoint : INT;
	//Alarm active for HMI
	{attribute 'OPC.UA.DA' :='1'}
	popa_0081_pt_3241_a_low_active : BOOL;
	//Analog Alarm Setpoint
	{attribute 'OPC.UA.DA' :='1'}
	popa_0081_pt_3241_a_low_setpoint : REAL;
	//Alarm enable
	{attribute 'OPC.UA.DA' :='1'}
	popa_0081_pt_3241_a_low_enable: BOOL;
	
	//Alarm Priority setpoint
	{attribute 'OPC.UA.DA' :='1'}
	popa_0081_pt_3241_a_high_priority : INT;
	//Alarm delay setpoint(seconds)
	{attribute 'OPC.UA.DA' :='1'}
	popa_0081_pt_3241_a_high_delay_setpoint : INT;
	//Alarm active for HMI
	{attribute 'OPC.UA.DA' :='1'}
	popa_0081_pt_3241_a_high_active : BOOL;
	//Analog Alarm Setpoint
	{attribute 'OPC.UA.DA' :='1'}
	popa_0081_pt_3241_a_high_setpoint : REAL;
	//Alarm enable
	{attribute 'OPC.UA.DA' :='1'}
	popa_0081_pt_3241_a_high_enable: BOOL;
	
	//Alarm Priority setpoint
	{attribute 'OPC.UA.DA' :='1'}
	popa_0081_pt_3241_a_high_high_priority : INT;
	//Alarm delay setpoint(seconds)
	{attribute 'OPC.UA.DA' :='1'}
	popa_0081_pt_3241_a_high_high_delay_setpoint : INT;
	//Alarm active for HMI
	{attribute 'OPC.UA.DA' :='1'}
	popa_0081_pt_3241_a_high_high_active : BOOL;
	//Analog Alarm Setpoint
	{attribute 'OPC.UA.DA' :='1'}
	popa_0081_pt_3241_a_high_high_setpoint : REAL;
	//Alarm enable
	{attribute 'OPC.UA.DA' :='1'}
	popa_0081_pt_3241_a_high_high_enable: BOOL;
	
	
	//Raw Min value for analog input
	{attribute 'OPC.UA.DA' :='1'}
	popa_0081_pt_3241_a_raw_min : REAL :=0;
	//Raw max value for analog input
	{attribute 'OPC.UA.DA' :='1'}
	popa_0081_pt_3241_a_raw_max : REAL :=32767;
	//EU Min value for analog input
	{attribute 'OPC.UA.DA' :='1'}
	popa_0081_pt_3241_a_eu_min : REAL;
	//EU Max value for analog input
	{attribute 'OPC.UA.DA' :='1'}
	popa_0081_pt_3241_a_eu_max : REAL;
	//Filter factor value for analog input
	{attribute 'OPC.UA.DA' :='1'}
	popa_0081_pt_3241_a_filter_factor : REAL;
	//Scaled value for analog input
	{attribute 'OPC.UA.DA' :='1'}
	popa_0081_pt_3241_a_scaled_value : REAL;
	
	//---pt_3341-----------------------------------------------------------------------------------------------------------------------
	//Alarm Priority setpoint
	{attribute 'OPC.UA.DA' :='1'}
	popa_0081_pt_3341_a_low_low_priority : INT;
	//Alarm delay setpoint(seconds)
	{attribute 'OPC.UA.DA' :='1'}
	popa_0081_pt_3341_a_low_low_delay_setpoint : INT;
	//Alarm active for HMI
	{attribute 'OPC.UA.DA' :='1'}
	popa_0081_pt_3341_a_low_low_active : BOOL;
	//Analog Alarm Setpoint
	{attribute 'OPC.UA.DA' :='1'}
	popa_0081_pt_3341_a_low_low_setpoint : REAL;
	//Alarm enable
	{attribute 'OPC.UA.DA' :='1'}
	popa_0081_pt_3341_a_low_low_enable: BOOL;
	
	//Alarm Priority setpoint
	{attribute 'OPC.UA.DA' :='1'}
	popa_0081_pt_3341_a_low_priority : INT;
	//Alarm delay setpoint(seconds)
	{attribute 'OPC.UA.DA' :='1'}
	popa_0081_pt_3341_a_low_delay_setpoint : INT;
	//Alarm active for HMI
	{attribute 'OPC.UA.DA' :='1'}
	popa_0081_pt_3341_a_low_active : BOOL;
	//Analog Alarm Setpoint
	{attribute 'OPC.UA.DA' :='1'}
	popa_0081_pt_3341_a_low_setpoint : REAL;
	//Alarm enable
	{attribute 'OPC.UA.DA' :='1'}
	popa_0081_pt_3341_a_low_enable: BOOL;
	
	//Alarm Priority setpoint
	{attribute 'OPC.UA.DA' :='1'}
	popa_0081_pt_3341_a_high_priority : INT;
	//Alarm delay setpoint(seconds)
	{attribute 'OPC.UA.DA' :='1'}
	popa_0081_pt_3341_a_high_delay_setpoint : INT;
	//Alarm active for HMI
	{attribute 'OPC.UA.DA' :='1'}
	popa_0081_pt_3341_a_high_active : BOOL;
	//Analog Alarm Setpoint
	{attribute 'OPC.UA.DA' :='1'}
	popa_0081_pt_3341_a_high_setpoint : REAL;
	//Alarm enable
	{attribute 'OPC.UA.DA' :='1'}
	popa_0081_pt_3341_a_high_enable: BOOL;
	
	//Alarm Priority setpoint
	{attribute 'OPC.UA.DA' :='1'}
	popa_0081_pt_3341_a_high_high_priority : INT;
	//Alarm delay setpoint(seconds)
	{attribute 'OPC.UA.DA' :='1'}
	popa_0081_pt_3341_a_high_high_delay_setpoint : INT;
	//Alarm active for HMI
	{attribute 'OPC.UA.DA' :='1'}
	popa_0081_pt_3341_a_high_high_active : BOOL;
	//Analog Alarm Setpoint
	{attribute 'OPC.UA.DA' :='1'}
	popa_0081_pt_3341_a_high_high_setpoint : REAL;
	//Alarm enable
	{attribute 'OPC.UA.DA' :='1'}
	popa_0081_pt_3341_a_high_high_enable: BOOL;
	
	
	//Raw Min value for analog input
	{attribute 'OPC.UA.DA' :='1'}
	popa_0081_pt_3341_a_raw_min : REAL :=0;
	//Raw max value for analog input
	{attribute 'OPC.UA.DA' :='1'}
	popa_0081_pt_3341_a_raw_max : REAL :=32767;
	//EU Min value for analog input
	{attribute 'OPC.UA.DA' :='1'}
	popa_0081_pt_3341_a_eu_min : REAL;
	//EU Max value for analog input
	{attribute 'OPC.UA.DA' :='1'}
	popa_0081_pt_3341_a_eu_max : REAL;
	//Filter factor value for analog input
	{attribute 'OPC.UA.DA' :='1'}
	popa_0081_pt_3341_a_filter_factor : REAL;
	//Scaled value for analog input
	{attribute 'OPC.UA.DA' :='1'}
	popa_0081_pt_3341_a_scaled_value : REAL;
	
//---pt_3428-----------------------------------------------------------------------------------------------------------------------
	//Alarm Priority setpoint
	{attribute 'OPC.UA.DA' :='1'}
	popa_0091_pt_3428_a_low_low_priority : INT;
	//Alarm delay setpoint(seconds)
	{attribute 'OPC.UA.DA' :='1'}
	popa_0091_pt_3428_a_low_low_delay_setpoint : INT;
	//Alarm active for HMI
	{attribute 'OPC.UA.DA' :='1'}
	popa_0091_pt_3428_a_low_low_active : BOOL;
	//Analog Alarm Setpoint
	{attribute 'OPC.UA.DA' :='1'}
	popa_0091_pt_3428_a_low_low_setpoint : REAL;
	//Alarm enable
	{attribute 'OPC.UA.DA' :='1'}
	popa_0091_pt_3428_a_low_low_enable: BOOL;
	
	//Alarm Priority setpoint
	{attribute 'OPC.UA.DA' :='1'}
	popa_0091_pt_3428_a_low_priority : INT;
	//Alarm delay setpoint(seconds)
	{attribute 'OPC.UA.DA' :='1'}
	popa_0091_pt_3428_a_low_delay_setpoint : INT;
	//Alarm active for HMI
	{attribute 'OPC.UA.DA' :='1'}
	popa_0091_pt_3428_a_low_active : BOOL;
	//Analog Alarm Setpoint
	{attribute 'OPC.UA.DA' :='1'}
	popa_0091_pt_3428_a_low_setpoint : REAL;
	//Alarm enable
	{attribute 'OPC.UA.DA' :='1'}
	popa_0091_pt_3428_a_low_enable: BOOL;
	
	//Alarm Priority setpoint
	{attribute 'OPC.UA.DA' :='1'}
	popa_0091_pt_3428_a_high_priority : INT;
	//Alarm delay setpoint(seconds)
	{attribute 'OPC.UA.DA' :='1'}
	popa_0091_pt_3428_a_high_delay_setpoint : INT;
	//Alarm active for HMI
	{attribute 'OPC.UA.DA' :='1'}
	popa_0091_pt_3428_a_high_active : BOOL;
	//Analog Alarm Setpoint
	{attribute 'OPC.UA.DA' :='1'}
	popa_0091_pt_3428_a_high_setpoint : REAL;
	//Alarm enable
	{attribute 'OPC.UA.DA' :='1'}
	popa_0091_pt_3428_a_high_enable: BOOL;
	
	//Alarm Priority setpoint
	{attribute 'OPC.UA.DA' :='1'}
	popa_0091_pt_3428_a_high_high_priority : INT;
	//Alarm delay setpoint(seconds)
	{attribute 'OPC.UA.DA' :='1'}
	popa_0091_pt_3428_a_high_high_delay_setpoint : INT;
	//Alarm active for HMI
	{attribute 'OPC.UA.DA' :='1'}
	popa_0091_pt_3428_a_high_high_active : BOOL;
	//Analog Alarm Setpoint
	{attribute 'OPC.UA.DA' :='1'}
	popa_0091_pt_3428_a_high_high_setpoint : REAL;
	//Alarm enable
	{attribute 'OPC.UA.DA' :='1'}
	popa_0091_pt_3428_a_high_high_enable: BOOL;
	
	
	//Raw Min value for analog input
	{attribute 'OPC.UA.DA' :='1'}
	popa_0091_pt_3428_a_raw_min : REAL :=0;
	//Raw max value for analog input
	{attribute 'OPC.UA.DA' :='1'}
	popa_0091_pt_3428_a_raw_max : REAL :=32767;
	//EU Min value for analog input
	{attribute 'OPC.UA.DA' :='1'}
	popa_0091_pt_3428_a_eu_min : REAL;
	//EU Max value for analog input
	{attribute 'OPC.UA.DA' :='1'}
	popa_0091_pt_3428_a_eu_max : REAL;
	//Filter factor value for analog input
	{attribute 'OPC.UA.DA' :='1'}
	popa_0091_pt_3428_a_filter_factor : REAL;
	//Scaled value for analog input
	{attribute 'OPC.UA.DA' :='1'}
	popa_0091_pt_3428_a_scaled_value : REAL;
	
	//---pt_3414-----------------------------------------------------------------------------------------------------------------------
	//Alarm Priority setpoint
	{attribute 'OPC.UA.DA' :='1'}
	popa_0091_pt_3414_a_low_low_priority : INT;
	//Alarm delay setpoint(seconds)
	{attribute 'OPC.UA.DA' :='1'}
	popa_0091_pt_3414_a_low_low_delay_setpoint : INT;
	//Alarm active for HMI
	{attribute 'OPC.UA.DA' :='1'}
	popa_0091_pt_3414_a_low_low_active : BOOL;
	//Analog Alarm Setpoint
	{attribute 'OPC.UA.DA' :='1'}
	popa_0091_pt_3414_a_low_low_setpoint : REAL;
	//Alarm enable
	{attribute 'OPC.UA.DA' :='1'}
	popa_0091_pt_3414_a_low_low_enable: BOOL;
	
	//Alarm Priority setpoint
	{attribute 'OPC.UA.DA' :='1'}
	popa_0091_pt_3414_a_low_priority : INT;
	//Alarm delay setpoint(seconds)
	{attribute 'OPC.UA.DA' :='1'}
	popa_0091_pt_3414_a_low_delay_setpoint : INT;
	//Alarm active for HMI
	{attribute 'OPC.UA.DA' :='1'}
	popa_0091_pt_3414_a_low_active : BOOL;
	//Analog Alarm Setpoint
	{attribute 'OPC.UA.DA' :='1'}
	popa_0091_pt_3414_a_low_setpoint : REAL;
	//Alarm enable
	{attribute 'OPC.UA.DA' :='1'}
	popa_0091_pt_3414_a_low_enable: BOOL;
	
	//Alarm Priority setpoint
	{attribute 'OPC.UA.DA' :='1'}
	popa_0091_pt_3414_a_high_priority : INT;
	//Alarm delay setpoint(seconds)
	{attribute 'OPC.UA.DA' :='1'}
	popa_0091_pt_3414_a_high_delay_setpoint : INT;
	//Alarm active for HMI
	{attribute 'OPC.UA.DA' :='1'}
	popa_0091_pt_3414_a_high_active : BOOL;
	//Analog Alarm Setpoint
	{attribute 'OPC.UA.DA' :='1'}
	popa_0091_pt_3414_a_high_setpoint : REAL;
	//Alarm enable
	{attribute 'OPC.UA.DA' :='1'}
	popa_0091_pt_3414_a_high_enable: BOOL;
	
	//Alarm Priority setpoint
	{attribute 'OPC.UA.DA' :='1'}
	popa_0091_pt_3414_a_high_high_priority : INT;
	//Alarm delay setpoint(seconds)
	{attribute 'OPC.UA.DA' :='1'}
	popa_0091_pt_3414_a_high_high_delay_setpoint : INT;
	//Alarm active for HMI
	{attribute 'OPC.UA.DA' :='1'}
	popa_0091_pt_3414_a_high_high_active : BOOL;
	//Analog Alarm Setpoint
	{attribute 'OPC.UA.DA' :='1'}
	popa_0091_pt_3414_a_high_high_setpoint : REAL;
	//Alarm enable
	{attribute 'OPC.UA.DA' :='1'}
	popa_0091_pt_3414_a_high_high_enable: BOOL;
	
	
	//Raw Min value for analog input
	{attribute 'OPC.UA.DA' :='1'}
	popa_0091_pt_3414_a_raw_min : REAL :=0;
	//Raw max value for analog input
	{attribute 'OPC.UA.DA' :='1'}
	popa_0091_pt_3414_a_raw_max : REAL :=32767;
	//EU Min value for analog input
	{attribute 'OPC.UA.DA' :='1'}
	popa_0091_pt_3414_a_eu_min : REAL;
	//EU Max value for analog input
	{attribute 'OPC.UA.DA' :='1'}
	popa_0091_pt_3414_a_eu_max : REAL;
	//Filter factor value for analog input
	{attribute 'OPC.UA.DA' :='1'}
	popa_0091_pt_3414_a_filter_factor : REAL;
	//Scaled value for analog input
	{attribute 'OPC.UA.DA' :='1'}
	popa_0091_pt_3414_a_scaled_value : REAL;
	
	//---tt_3118-----------------------------------------------------------------------------------------------------------------------
	//Alarm Priority setpoint
	{attribute 'OPC.UA.DA' :='1'}
	popa_0081_tt_3118_a_low_low_priority : INT;
	//Alarm delay setpoint(seconds)
	{attribute 'OPC.UA.DA' :='1'}
	popa_0081_tt_3118_a_low_low_delay_setpoint : INT;
	//Alarm active for HMI
	{attribute 'OPC.UA.DA' :='1'}
	popa_0081_tt_3118_a_low_low_active : BOOL;
	//Analog Alarm Setpoint
	{attribute 'OPC.UA.DA' :='1'}
	popa_0081_tt_3118_a_low_low_setpoint : REAL;
	//Alarm enable
	{attribute 'OPC.UA.DA' :='1'}
	popa_0081_tt_3118_a_low_low_enable: BOOL;
	
	//Alarm Priority setpoint
	{attribute 'OPC.UA.DA' :='1'}
	popa_0081_tt_3118_a_low_priority : INT;
	//Alarm delay setpoint(seconds)
	{attribute 'OPC.UA.DA' :='1'}
	popa_0081_tt_3118_a_low_delay_setpoint : INT;
	//Alarm active for HMI
	{attribute 'OPC.UA.DA' :='1'}
	popa_0081_tt_3118_a_low_active : BOOL;
	//Analog Alarm Setpoint
	{attribute 'OPC.UA.DA' :='1'}
	popa_0081_tt_3118_a_low_setpoint : REAL;
	//Alarm enable
	{attribute 'OPC.UA.DA' :='1'}
	popa_0081_tt_3118_a_low_enable: BOOL;
	
	//Alarm Priority setpoint
	{attribute 'OPC.UA.DA' :='1'}
	popa_0081_tt_3118_a_high_priority : INT;
	//Alarm delay setpoint(seconds)
	{attribute 'OPC.UA.DA' :='1'}
	popa_0081_tt_3118_a_high_delay_setpoint : INT;
	//Alarm active for HMI
	{attribute 'OPC.UA.DA' :='1'}
	popa_0081_tt_3118_a_high_active : BOOL;
	//Analog Alarm Setpoint
	{attribute 'OPC.UA.DA' :='1'}
	popa_0081_tt_3118_a_high_setpoint : REAL;
	//Alarm enable
	{attribute 'OPC.UA.DA' :='1'}
	popa_0081_tt_3118_a_high_enable: BOOL;
	
	//Alarm Priority setpoint
	{attribute 'OPC.UA.DA' :='1'}
	popa_0081_tt_3118_a_high_high_priority : INT;
	//Alarm delay setpoint(seconds)
	{attribute 'OPC.UA.DA' :='1'}
	popa_0081_tt_3118_a_high_high_delay_setpoint : INT;
	//Alarm active for HMI
	{attribute 'OPC.UA.DA' :='1'}
	popa_0081_tt_3118_a_high_high_active : BOOL;
	//Analog Alarm Setpoint
	{attribute 'OPC.UA.DA' :='1'}
	popa_0081_tt_3118_a_high_high_setpoint : REAL;
	//Alarm enable
	{attribute 'OPC.UA.DA' :='1'}
	popa_0081_tt_3118_a_high_high_enable: BOOL;
	
	
	//Raw Min value for analog input
	{attribute 'OPC.UA.DA' :='1'}
	popa_0081_tt_3118_a_raw_min : REAL :=0;
	//Raw max value for analog input
	{attribute 'OPC.UA.DA' :='1'}
	popa_0081_tt_3118_a_raw_max : REAL :=32767;
	//EU Min value for analog input
	{attribute 'OPC.UA.DA' :='1'}
	popa_0081_tt_3118_a_eu_min : REAL;
	//EU Max value for analog input
	{attribute 'OPC.UA.DA' :='1'}
	popa_0081_tt_3118_a_eu_max : REAL;
	//Filter factor value for analog input
	{attribute 'OPC.UA.DA' :='1'}
	popa_0081_tt_3118_a_filter_factor : REAL;
	//Scaled value for analog input
	{attribute 'OPC.UA.DA' :='1'}
	popa_0081_tt_3118_a_scaled_value : REAL;
	
	//---tt_3218-----------------------------------------------------------------------------------------------------------------------
	//Alarm Priority setpoint
	{attribute 'OPC.UA.DA' :='1'}
	popa_0081_tt_3218_a_low_low_priority : INT;
	//Alarm delay setpoint(seconds)
	{attribute 'OPC.UA.DA' :='1'}
	popa_0081_tt_3218_a_low_low_delay_setpoint : INT;
	//Alarm active for HMI
	{attribute 'OPC.UA.DA' :='1'}
	popa_0081_tt_3218_a_low_low_active : BOOL;
	//Analog Alarm Setpoint
	{attribute 'OPC.UA.DA' :='1'}
	popa_0081_tt_3218_a_low_low_setpoint : REAL;
	//Alarm enable
	{attribute 'OPC.UA.DA' :='1'}
	popa_0081_tt_3218_a_low_low_enable: BOOL;
	
	//Alarm Priority setpoint
	{attribute 'OPC.UA.DA' :='1'}
	popa_0081_tt_3218_a_low_priority : INT;
	//Alarm delay setpoint(seconds)
	{attribute 'OPC.UA.DA' :='1'}
	popa_0081_tt_3218_a_low_delay_setpoint : INT;
	//Alarm active for HMI
	{attribute 'OPC.UA.DA' :='1'}
	popa_0081_tt_3218_a_low_active : BOOL;
	//Analog Alarm Setpoint
	{attribute 'OPC.UA.DA' :='1'}
	popa_0081_tt_3218_a_low_setpoint : REAL;
	//Alarm enable
	{attribute 'OPC.UA.DA' :='1'}
	popa_0081_tt_3218_a_low_enable: BOOL;
	
	//Alarm Priority setpoint
	{attribute 'OPC.UA.DA' :='1'}
	popa_0081_tt_3218_a_high_priority : INT;
	//Alarm delay setpoint(seconds)
	{attribute 'OPC.UA.DA' :='1'}
	popa_0081_tt_3218_a_high_delay_setpoint : INT;
	//Alarm active for HMI
	{attribute 'OPC.UA.DA' :='1'}
	popa_0081_tt_3218_a_high_active : BOOL;
	//Analog Alarm Setpoint
	{attribute 'OPC.UA.DA' :='1'}
	popa_0081_tt_3218_a_high_setpoint : REAL;
	//Alarm enable
	{attribute 'OPC.UA.DA' :='1'}
	popa_0081_tt_3218_a_high_enable: BOOL;
	
	//Alarm Priority setpoint
	{attribute 'OPC.UA.DA' :='1'}
	popa_0081_tt_3218_a_high_high_priority : INT;
	//Alarm delay setpoint(seconds)
	{attribute 'OPC.UA.DA' :='1'}
	popa_0081_tt_3218_a_high_high_delay_setpoint : INT;
	//Alarm active for HMI
	{attribute 'OPC.UA.DA' :='1'}
	popa_0081_tt_3218_a_high_high_active : BOOL;
	//Analog Alarm Setpoint
	{attribute 'OPC.UA.DA' :='1'}
	popa_0081_tt_3218_a_high_high_setpoint : REAL;
	//Alarm enable
	{attribute 'OPC.UA.DA' :='1'}
	popa_0081_tt_3218_a_high_high_enable: BOOL;
	
	
	//Raw Min value for analog input
	{attribute 'OPC.UA.DA' :='1'}
	popa_0081_tt_3218_a_raw_min : REAL :=0;
	//Raw max value for analog input
	{attribute 'OPC.UA.DA' :='1'}
	popa_0081_tt_3218_a_raw_max : REAL :=32767;
	//EU Min value for analog input
	{attribute 'OPC.UA.DA' :='1'}
	popa_0081_tt_3218_a_eu_min : REAL;
	//EU Max value for analog input
	{attribute 'OPC.UA.DA' :='1'}
	popa_0081_tt_3218_a_eu_max : REAL;
	//Filter factor value for analog input
	{attribute 'OPC.UA.DA' :='1'}
	popa_0081_tt_3218_a_filter_factor : REAL;
	//Scaled value for analog input
	{attribute 'OPC.UA.DA' :='1'}
	popa_0081_tt_3218_a_scaled_value : REAL;
	
	//---tt_3318-----------------------------------------------------------------------------------------------------------------------
	//Alarm Priority setpoint
	{attribute 'OPC.UA.DA' :='1'}
	popa_0081_tt_3318_a_low_low_priority : INT;
	//Alarm delay setpoint(seconds)
	{attribute 'OPC.UA.DA' :='1'}
	popa_0081_tt_3318_a_low_low_delay_setpoint : INT;
	//Alarm active for HMI
	{attribute 'OPC.UA.DA' :='1'}
	popa_0081_tt_3318_a_low_low_active : BOOL;
	//Analog Alarm Setpoint
	{attribute 'OPC.UA.DA' :='1'}
	popa_0081_tt_3318_a_low_low_setpoint : REAL;
	//Alarm enable
	{attribute 'OPC.UA.DA' :='1'}
	popa_0081_tt_3318_a_low_low_enable: BOOL;
	
	//Alarm Priority setpoint
	{attribute 'OPC.UA.DA' :='1'}
	popa_0081_tt_3318_a_low_priority : INT;
	//Alarm delay setpoint(seconds)
	{attribute 'OPC.UA.DA' :='1'}
	popa_0081_tt_3318_a_low_delay_setpoint : INT;
	//Alarm active for HMI
	{attribute 'OPC.UA.DA' :='1'}
	popa_0081_tt_3318_a_low_active : BOOL;
	//Analog Alarm Setpoint
	{attribute 'OPC.UA.DA' :='1'}
	popa_0081_tt_3318_a_low_setpoint : REAL;
	//Alarm enable
	{attribute 'OPC.UA.DA' :='1'}
	popa_0081_tt_3318_a_low_enable: BOOL;
	
	//Alarm Priority setpoint
	{attribute 'OPC.UA.DA' :='1'}
	popa_0081_tt_3318_a_high_priority : INT;
	//Alarm delay setpoint(seconds)
	{attribute 'OPC.UA.DA' :='1'}
	popa_0081_tt_3318_a_high_delay_setpoint : INT;
	//Alarm active for HMI
	{attribute 'OPC.UA.DA' :='1'}
	popa_0081_tt_3318_a_high_active : BOOL;
	//Analog Alarm Setpoint
	{attribute 'OPC.UA.DA' :='1'}
	popa_0081_tt_3318_a_high_setpoint : REAL;
	//Alarm enable
	{attribute 'OPC.UA.DA' :='1'}
	popa_0081_tt_3318_a_high_enable: BOOL;
	
	//Alarm Priority setpoint
	{attribute 'OPC.UA.DA' :='1'}
	popa_0081_tt_3318_a_high_high_priority : INT;
	//Alarm delay setpoint(seconds)
	{attribute 'OPC.UA.DA' :='1'}
	popa_0081_tt_3318_a_high_high_delay_setpoint : INT;
	//Alarm active for HMI
	{attribute 'OPC.UA.DA' :='1'}
	popa_0081_tt_3318_a_high_high_active : BOOL;
	//Analog Alarm Setpoint
	{attribute 'OPC.UA.DA' :='1'}
	popa_0081_tt_3318_a_high_high_setpoint : REAL;
	//Alarm enable
	{attribute 'OPC.UA.DA' :='1'}
	popa_0081_tt_3318_a_high_high_enable: BOOL;
	
	
	//Raw Min value for analog input
	{attribute 'OPC.UA.DA' :='1'}
	popa_0081_tt_3318_a_raw_min : REAL :=0;
	//Raw max value for analog input
	{attribute 'OPC.UA.DA' :='1'}
	popa_0081_tt_3318_a_raw_max : REAL :=32767;
	//EU Min value for analog input
	{attribute 'OPC.UA.DA' :='1'}
	popa_0081_tt_3318_a_eu_min : REAL;
	//EU Max value for analog input
	{attribute 'OPC.UA.DA' :='1'}
	popa_0081_tt_3318_a_eu_max : REAL;
	//Filter factor value for analog input
	{attribute 'OPC.UA.DA' :='1'}
	popa_0081_tt_3318_a_filter_factor : REAL;
	//Scaled value for analog input
	{attribute 'OPC.UA.DA' :='1'}
	popa_0081_tt_3318_a_scaled_value : REAL;
	
	//---tt_3140-----------------------------------------------------------------------------------------------------------------------
	//Alarm Priority setpoint
	{attribute 'OPC.UA.DA' :='1'}
	popa_0081_tt_3140_a_low_low_priority : INT;
	//Alarm delay setpoint(seconds)
	{attribute 'OPC.UA.DA' :='1'}
	popa_0081_tt_3140_a_low_low_delay_setpoint : INT;
	//Alarm active for HMI
	{attribute 'OPC.UA.DA' :='1'}
	popa_0081_tt_3140_a_low_low_active : BOOL;
	//Analog Alarm Setpoint
	{attribute 'OPC.UA.DA' :='1'}
	popa_0081_tt_3140_a_low_low_setpoint : REAL;
	//Alarm enable
	{attribute 'OPC.UA.DA' :='1'}
	popa_0081_tt_3140_a_low_low_enable: BOOL;
	
	//Alarm Priority setpoint
	{attribute 'OPC.UA.DA' :='1'}
	popa_0081_tt_3140_a_low_priority : INT;
	//Alarm delay setpoint(seconds)
	{attribute 'OPC.UA.DA' :='1'}
	popa_0081_tt_3140_a_low_delay_setpoint : INT;
	//Alarm active for HMI
	{attribute 'OPC.UA.DA' :='1'}
	popa_0081_tt_3140_a_low_active : BOOL;
	//Analog Alarm Setpoint
	{attribute 'OPC.UA.DA' :='1'}
	popa_0081_tt_3140_a_low_setpoint : REAL;
	//Alarm enable
	{attribute 'OPC.UA.DA' :='1'}
	popa_0081_tt_3140_a_low_enable: BOOL;
	
	//Alarm Priority setpoint
	{attribute 'OPC.UA.DA' :='1'}
	popa_0081_tt_3140_a_high_priority : INT;
	//Alarm delay setpoint(seconds)
	{attribute 'OPC.UA.DA' :='1'}
	popa_0081_tt_3140_a_high_delay_setpoint : INT;
	//Alarm active for HMI
	{attribute 'OPC.UA.DA' :='1'}
	popa_0081_tt_3140_a_high_active : BOOL;
	//Analog Alarm Setpoint
	{attribute 'OPC.UA.DA' :='1'}
	popa_0081_tt_3140_a_high_setpoint : REAL;
	//Alarm enable
	{attribute 'OPC.UA.DA' :='1'}
	popa_0081_tt_3140_a_high_enable: BOOL;
	
	//Alarm Priority setpoint
	{attribute 'OPC.UA.DA' :='1'}
	popa_0081_tt_3140_a_high_high_priority : INT;
	//Alarm delay setpoint(seconds)
	{attribute 'OPC.UA.DA' :='1'}
	popa_0081_tt_3140_a_high_high_delay_setpoint : INT;
	//Alarm active for HMI
	{attribute 'OPC.UA.DA' :='1'}
	popa_0081_tt_3140_a_high_high_active : BOOL;
	//Analog Alarm Setpoint
	{attribute 'OPC.UA.DA' :='1'}
	popa_0081_tt_3140_a_high_high_setpoint : REAL;
	//Alarm enable
	{attribute 'OPC.UA.DA' :='1'}
	popa_0081_tt_3140_a_high_high_enable: BOOL;
	
	
	//Raw Min value for analog input
	{attribute 'OPC.UA.DA' :='1'}
	popa_0081_tt_3140_a_raw_min : REAL :=0;
	//Raw max value for analog input
	{attribute 'OPC.UA.DA' :='1'}
	popa_0081_tt_3140_a_raw_max : REAL :=32767;
	//EU Min value for analog input
	{attribute 'OPC.UA.DA' :='1'}
	popa_0081_tt_3140_a_eu_min : REAL;
	//EU Max value for analog input
	{attribute 'OPC.UA.DA' :='1'}
	popa_0081_tt_3140_a_eu_max : REAL;
	//Filter factor value for analog input
	{attribute 'OPC.UA.DA' :='1'}
	popa_0081_tt_3140_a_filter_factor : REAL;
	//Scaled value for analog input
	{attribute 'OPC.UA.DA' :='1'}
	popa_0081_tt_3140_a_scaled_value : REAL;
	
	//---tt_3240-----------------------------------------------------------------------------------------------------------------------
	//Alarm Priority setpoint
	{attribute 'OPC.UA.DA' :='1'}
	popa_0081_tt_3240_a_low_low_priority : INT;
	//Alarm delay setpoint(seconds)
	{attribute 'OPC.UA.DA' :='1'}
	popa_0081_tt_3240_a_low_low_delay_setpoint : INT;
	//Alarm active for HMI
	{attribute 'OPC.UA.DA' :='1'}
	popa_0081_tt_3240_a_low_low_active : BOOL;
	//Analog Alarm Setpoint
	{attribute 'OPC.UA.DA' :='1'}
	popa_0081_tt_3240_a_low_low_setpoint : REAL;
	//Alarm enable
	{attribute 'OPC.UA.DA' :='1'}
	popa_0081_tt_3240_a_low_low_enable: BOOL;
	
	//Alarm Priority setpoint
	{attribute 'OPC.UA.DA' :='1'}
	popa_0081_tt_3240_a_low_priority : INT;
	//Alarm delay setpoint(seconds)
	{attribute 'OPC.UA.DA' :='1'}
	popa_0081_tt_3240_a_low_delay_setpoint : INT;
	//Alarm active for HMI
	{attribute 'OPC.UA.DA' :='1'}
	popa_0081_tt_3240_a_low_active : BOOL;
	//Analog Alarm Setpoint
	{attribute 'OPC.UA.DA' :='1'}
	popa_0081_tt_3240_a_low_setpoint : REAL;
	//Alarm enable
	{attribute 'OPC.UA.DA' :='1'}
	popa_0081_tt_3240_a_low_enable: BOOL;
	
	//Alarm Priority setpoint
	{attribute 'OPC.UA.DA' :='1'}
	popa_0081_tt_3240_a_high_priority : INT;
	//Alarm delay setpoint(seconds)
	{attribute 'OPC.UA.DA' :='1'}
	popa_0081_tt_3240_a_high_delay_setpoint : INT;
	//Alarm active for HMI
	{attribute 'OPC.UA.DA' :='1'}
	popa_0081_tt_3240_a_high_active : BOOL;
	//Analog Alarm Setpoint
	{attribute 'OPC.UA.DA' :='1'}
	popa_0081_tt_3240_a_high_setpoint : REAL;
	//Alarm enable
	{attribute 'OPC.UA.DA' :='1'}
	popa_0081_tt_3240_a_high_enable: BOOL;
	
	//Alarm Priority setpoint
	{attribute 'OPC.UA.DA' :='1'}
	popa_0081_tt_3240_a_high_high_priority : INT;
	//Alarm delay setpoint(seconds)
	{attribute 'OPC.UA.DA' :='1'}
	popa_0081_tt_3240_a_high_high_delay_setpoint : INT;
	//Alarm active for HMI
	{attribute 'OPC.UA.DA' :='1'}
	popa_0081_tt_3240_a_high_high_active : BOOL;
	//Analog Alarm Setpoint
	{attribute 'OPC.UA.DA' :='1'}
	popa_0081_tt_3240_a_high_high_setpoint : REAL;
	//Alarm enable
	{attribute 'OPC.UA.DA' :='1'}
	popa_0081_tt_3240_a_high_high_enable: BOOL;
	
	
	//Raw Min value for analog input
	{attribute 'OPC.UA.DA' :='1'}
	popa_0081_tt_3240_a_raw_min : REAL :=0;
	//Raw max value for analog input
	{attribute 'OPC.UA.DA' :='1'}
	popa_0081_tt_3240_a_raw_max : REAL :=32767;
	//EU Min value for analog input
	{attribute 'OPC.UA.DA' :='1'}
	popa_0081_tt_3240_a_eu_min : REAL;
	//EU Max value for analog input
	{attribute 'OPC.UA.DA' :='1'}
	popa_0081_tt_3240_a_eu_max : REAL;
	//Filter factor value for analog input
	{attribute 'OPC.UA.DA' :='1'}
	popa_0081_tt_3240_a_filter_factor : REAL;
	//Scaled value for analog input
	{attribute 'OPC.UA.DA' :='1'}
	popa_0081_tt_3240_a_scaled_value : REAL;
	
	//---tt_3340-----------------------------------------------------------------------------------------------------------------------
	//Alarm Priority setpoint
	{attribute 'OPC.UA.DA' :='1'}
	popa_0081_tt_3340_a_low_low_priority : INT;
	//Alarm delay setpoint(seconds)
	{attribute 'OPC.UA.DA' :='1'}
	popa_0081_tt_3340_a_low_low_delay_setpoint : INT;
	//Alarm active for HMI
	{attribute 'OPC.UA.DA' :='1'}
	popa_0081_tt_3340_a_low_low_active : BOOL;
	//Analog Alarm Setpoint
	{attribute 'OPC.UA.DA' :='1'}
	popa_0081_tt_3340_a_low_low_setpoint : REAL;
	//Alarm enable
	{attribute 'OPC.UA.DA' :='1'}
	popa_0081_tt_3340_a_low_low_enable: BOOL;
	
	//Alarm Priority setpoint
	{attribute 'OPC.UA.DA' :='1'}
	popa_0081_tt_3340_a_low_priority : INT;
	//Alarm delay setpoint(seconds)
	{attribute 'OPC.UA.DA' :='1'}
	popa_0081_tt_3340_a_low_delay_setpoint : INT;
	//Alarm active for HMI
	{attribute 'OPC.UA.DA' :='1'}
	popa_0081_tt_3340_a_low_active : BOOL;
	//Analog Alarm Setpoint
	{attribute 'OPC.UA.DA' :='1'}
	popa_0081_tt_3340_a_low_setpoint : REAL;
	//Alarm enable
	{attribute 'OPC.UA.DA' :='1'}
	popa_0081_tt_3340_a_low_enable: BOOL;
	
	//Alarm Priority setpoint
	{attribute 'OPC.UA.DA' :='1'}
	popa_0081_tt_3340_a_high_priority : INT;
	//Alarm delay setpoint(seconds)
	{attribute 'OPC.UA.DA' :='1'}
	popa_0081_tt_3340_a_high_delay_setpoint : INT;
	//Alarm active for HMI
	{attribute 'OPC.UA.DA' :='1'}
	popa_0081_tt_3340_a_high_active : BOOL;
	//Analog Alarm Setpoint
	{attribute 'OPC.UA.DA' :='1'}
	popa_0081_tt_3340_a_high_setpoint : REAL;
	//Alarm enable
	{attribute 'OPC.UA.DA' :='1'}
	popa_0081_tt_3340_a_high_enable: BOOL;
	
	//Alarm Priority setpoint
	{attribute 'OPC.UA.DA' :='1'}
	popa_0081_tt_3340_a_high_high_priority : INT;
	//Alarm delay setpoint(seconds)
	{attribute 'OPC.UA.DA' :='1'}
	popa_0081_tt_3340_a_high_high_delay_setpoint : INT;
	//Alarm active for HMI
	{attribute 'OPC.UA.DA' :='1'}
	popa_0081_tt_3340_a_high_high_active : BOOL;
	//Analog Alarm Setpoint
	{attribute 'OPC.UA.DA' :='1'}
	popa_0081_tt_3340_a_high_high_setpoint : REAL;
	//Alarm enable
	{attribute 'OPC.UA.DA' :='1'}
	popa_0081_tt_3340_a_high_high_enable: BOOL;
	
	
	//Raw Min value for analog input
	{attribute 'OPC.UA.DA' :='1'}
	popa_0081_tt_3340_a_raw_min : REAL :=0;
	//Raw max value for analog input
	{attribute 'OPC.UA.DA' :='1'}
	popa_0081_tt_3340_a_raw_max : REAL :=32767;
	//EU Min value for analog input
	{attribute 'OPC.UA.DA' :='1'}
	popa_0081_tt_3340_a_eu_min : REAL;
	//EU Max value for analog input
	{attribute 'OPC.UA.DA' :='1'}
	popa_0081_tt_3340_a_eu_max : REAL;
	//Filter factor value for analog input
	{attribute 'OPC.UA.DA' :='1'}
	popa_0081_tt_3340_a_filter_factor : REAL;
	//Scaled value for analog input
	{attribute 'OPC.UA.DA' :='1'}
	popa_0081_tt_3340_a_scaled_value : REAL;
	
	//---tt_3432-----------------------------------------------------------------------------------------------------------------------
	//Alarm Priority setpoint
	{attribute 'OPC.UA.DA' :='1'}
	popa_0091_tt_3432_a_low_low_priority : INT;
	//Alarm delay setpoint(seconds)
	{attribute 'OPC.UA.DA' :='1'}
	popa_0091_tt_3432_a_low_low_delay_setpoint : INT;
	//Alarm active for HMI
	{attribute 'OPC.UA.DA' :='1'}
	popa_0091_tt_3432_a_low_low_active : BOOL;
	//Analog Alarm Setpoint
	{attribute 'OPC.UA.DA' :='1'}
	popa_0091_tt_3432_a_low_low_setpoint : REAL;
	//Alarm enable
	{attribute 'OPC.UA.DA' :='1'}
	popa_0091_tt_3432_a_low_low_enable: BOOL;
	
	//Alarm Priority setpoint
	{attribute 'OPC.UA.DA' :='1'}
	popa_0091_tt_3432_a_low_priority : INT;
	//Alarm delay setpoint(seconds)
	{attribute 'OPC.UA.DA' :='1'}
	popa_0091_tt_3432_a_low_delay_setpoint : INT;
	//Alarm active for HMI
	{attribute 'OPC.UA.DA' :='1'}
	popa_0091_tt_3432_a_low_active : BOOL;
	//Analog Alarm Setpoint
	{attribute 'OPC.UA.DA' :='1'}
	popa_0091_tt_3432_a_low_setpoint : REAL;
	//Alarm enable
	{attribute 'OPC.UA.DA' :='1'}
	popa_0091_tt_3432_a_low_enable: BOOL;
	
	//Alarm Priority setpoint
	{attribute 'OPC.UA.DA' :='1'}
	popa_0091_tt_3432_a_high_priority : INT;
	//Alarm delay setpoint(seconds)
	{attribute 'OPC.UA.DA' :='1'}
	popa_0091_tt_3432_a_high_delay_setpoint : INT;
	//Alarm active for HMI
	{attribute 'OPC.UA.DA' :='1'}
	popa_0091_tt_3432_a_high_active : BOOL;
	//Analog Alarm Setpoint
	{attribute 'OPC.UA.DA' :='1'}
	popa_0091_tt_3432_a_high_setpoint : REAL;
	//Alarm enable
	{attribute 'OPC.UA.DA' :='1'}
	popa_0091_tt_3432_a_high_enable: BOOL;
	
	//Alarm Priority setpoint
	{attribute 'OPC.UA.DA' :='1'}
	popa_0091_tt_3432_a_high_high_priority : INT;
	//Alarm delay setpoint(seconds)
	{attribute 'OPC.UA.DA' :='1'}
	popa_0091_tt_3432_a_high_high_delay_setpoint : INT;
	//Alarm active for HMI
	{attribute 'OPC.UA.DA' :='1'}
	popa_0091_tt_3432_a_high_high_active : BOOL;
	//Analog Alarm Setpoint
	{attribute 'OPC.UA.DA' :='1'}
	popa_0091_tt_3432_a_high_high_setpoint : REAL;
	//Alarm enable
	{attribute 'OPC.UA.DA' :='1'}
	popa_0091_tt_3432_a_high_high_enable: BOOL;
	
	
	//Raw Min value for analog input
	{attribute 'OPC.UA.DA' :='1'}
	popa_0091_tt_3432_a_raw_min : REAL :=0;
	//Raw max value for analog input
	{attribute 'OPC.UA.DA' :='1'}
	popa_0091_tt_3432_a_raw_max : REAL :=32767;
	//EU Min value for analog input
	{attribute 'OPC.UA.DA' :='1'}
	popa_0091_tt_3432_a_eu_min : REAL;
	//EU Max value for analog input
	{attribute 'OPC.UA.DA' :='1'}
	popa_0091_tt_3432_a_eu_max : REAL;
	//Filter factor value for analog input
	{attribute 'OPC.UA.DA' :='1'}
	popa_0091_tt_3432_a_filter_factor : REAL;
	//Scaled value for analog input
	{attribute 'OPC.UA.DA' :='1'}
	popa_0091_tt_3432_a_scaled_value : REAL;
	
END_VAR

// ---- GVLs/plccomms.TcGVL
{attribute 'qualified_only'}
VAR_GLOBAL PERSISTENT
	popa_0081_publish_real AT %Q* : ARRAY[0..99] OF REAL;
	popa_0081_publish_bool AT %Q* : ARRAY[0..99] OF BOOL;
	popa_supervisor_subscribe_real AT %I* : ARRAY[0..99] OF REAL;
	popa_supervisor_subscribe_bool AT %I* : ARRAY[0..99] OF BOOL;
END_VAR

// ---- POUs/example_loop_control.TcPOU
PROGRAM example_loop_control
VAR
	//Example run request for a starter motor.  This would be triggered by control loop logic
	u_3160_a_run_request : BOOL;
	
	//Example run request for a vfd motor.  This would be triggered by control loop logic
	u_3112_a_run_request : BOOL;
	//Example Speed Request for a vfd motor.  This would be set by control loop logic, normally a PID
	u_3112_a_speed_request : REAL;
	
	//Example position request for an analog valve.  This would be set by control loop logic, normally a PID
	av_3148_a_position_request : REAL;
	
	//Example open request for a digital valve.  This would be triggered by control loop logic
	nv_3372_a_open_request : BOOL;
END_VAR

// NETWORK 1

END_PROGRAM

// ---- POUs/general.TcPOU
PROGRAM general
VAR PERSISTENT
	//System date time function block
	system_date_time : date_time;
	//Daily reset bit, used throughout the program for any resets
	daily_reset : BOOL;
	//Alarm Acknoweldge unlatch timer
	alarm_ack_ton : ton;
	//Alarm Reset unlatch timer
	alarm_reset_ton : ton;
	//Alarm Ack and reset unlatch timer setpoint
	alarm_ack_unlatch_sp : TIME :=T#1S;
	
	//Always off bit
	always_off : BOOL := FALSE;
	
	//PLC States - move as needed
	ed_routine_idle : BOOL;
	ed_routine_cip : BOOL;
	ed_routine_manual : BOOL;
	ed_routine_maint : BOOL;
	ed_routine_stop : BOOL;
	ed_critical_stop : BOOL;
	
END_VAR

VAR
	//{attribute 'TcLinkTo' := 'TIID^Device 1 (EtherCAT)^Term 1 (EK1200)^Term 10 (EL2911)^StandardInputs^Standard Out Var 16'}
	twinsafe_safeout AT %I*: BOOL;
	
	//Linked manually
	twinsafe_status AT %I*: USINT;
	twinsafe_reset AT %Q*: BOOL;
	twinsafe_ack AT %Q*: BOOL;
	twinsafe_run AT %Q*: BOOL := TRUE;
	
	test_valve_position AT %I*: INT;
	
	
	test_valve: analog_scaling;
	test_nv_3110_open: BOOL;
	safety_reset_ton: TON;
	eng_test: BOOL;
	Safety_out: BOOL;
END_VAR
VAR // added by the converter: edge detectors and wires of the graphical bodies
    _rt1, _rt2, _rt3, _rt4, _rt5 : R_TRIG;
    _w1, _w2, _w3, _w4 : BOOL;
END_VAR

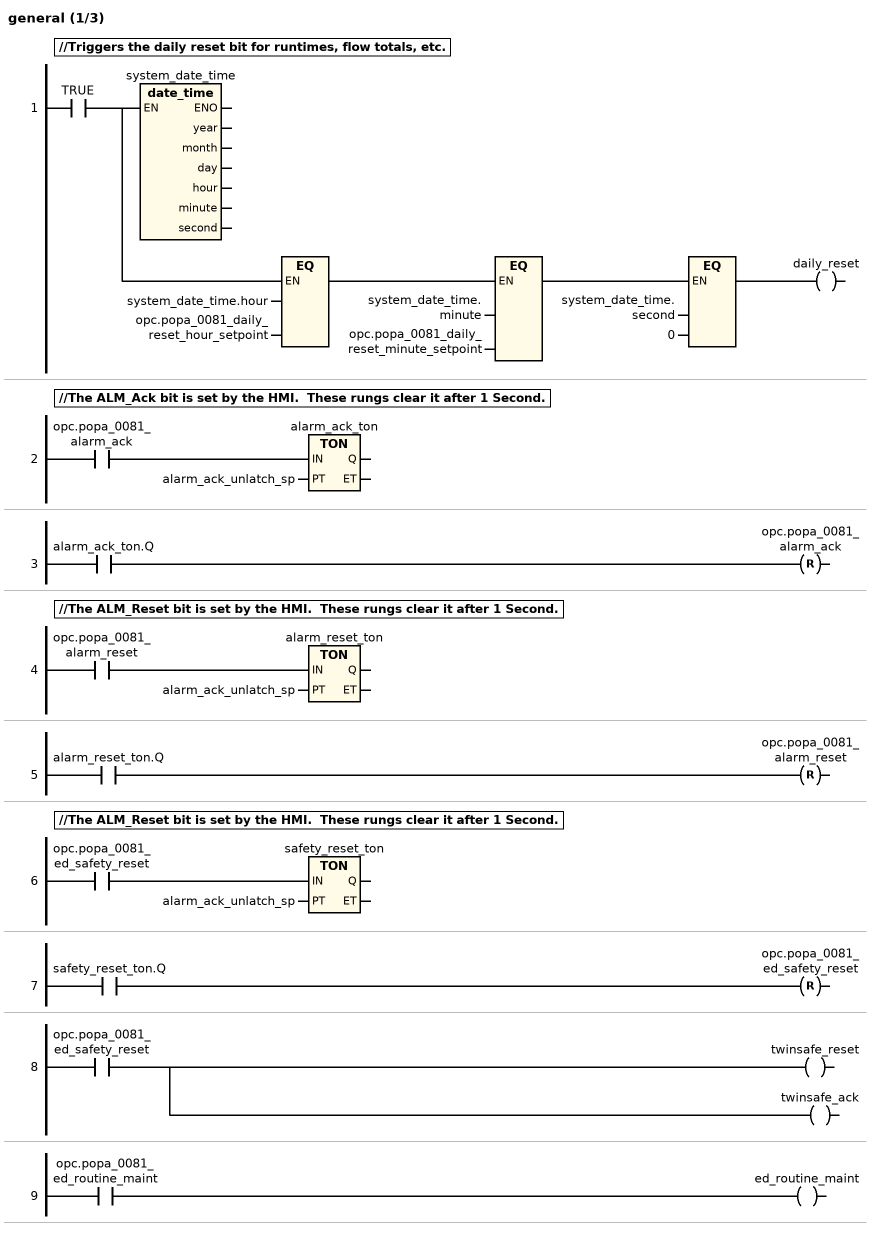
// NETWORK 1
// label: //Triggers the daily reset bit for runtimes, flow totals, etc.
system_date_time(); // date_time
daily_reset := system_date_time.hour = opc.popa_0081_daily_reset_hour_setpoint AND system_date_time.minute = opc.popa_0081_daily_reset_minute_setpoint AND system_date_time.second = 0;

// NETWORK 2
// label: //The ALM_Ack bit is set by the HMI.  These rungs clear it after 1 Second.
alarm_ack_ton(IN := opc.popa_0081_alarm_ack, PT := alarm_ack_unlatch_sp); // TON

// NETWORK 3
opc.popa_0081_alarm_ack R= alarm_ack_ton.Q;

// NETWORK 4
// label: //The ALM_Reset bit is set by the HMI.  These rungs clear it after 1 Second.
alarm_reset_ton(IN := opc.popa_0081_alarm_reset, PT := alarm_ack_unlatch_sp); // TON

// NETWORK 5
opc.popa_0081_alarm_reset R= alarm_reset_ton.Q;

// NETWORK 6
// label: //The ALM_Reset bit is set by the HMI.  These rungs clear it after 1 Second.
safety_reset_ton(IN := opc.popa_0081_ed_safety_reset, PT := alarm_ack_unlatch_sp); // TON

// NETWORK 7
opc.popa_0081_ed_safety_reset R= safety_reset_ton.Q;

// NETWORK 8
twinsafe_reset := opc.popa_0081_ed_safety_reset;
twinsafe_ack := opc.popa_0081_ed_safety_reset;

// NETWORK 9
ed_routine_maint := opc.popa_0081_ed_routine_maint;

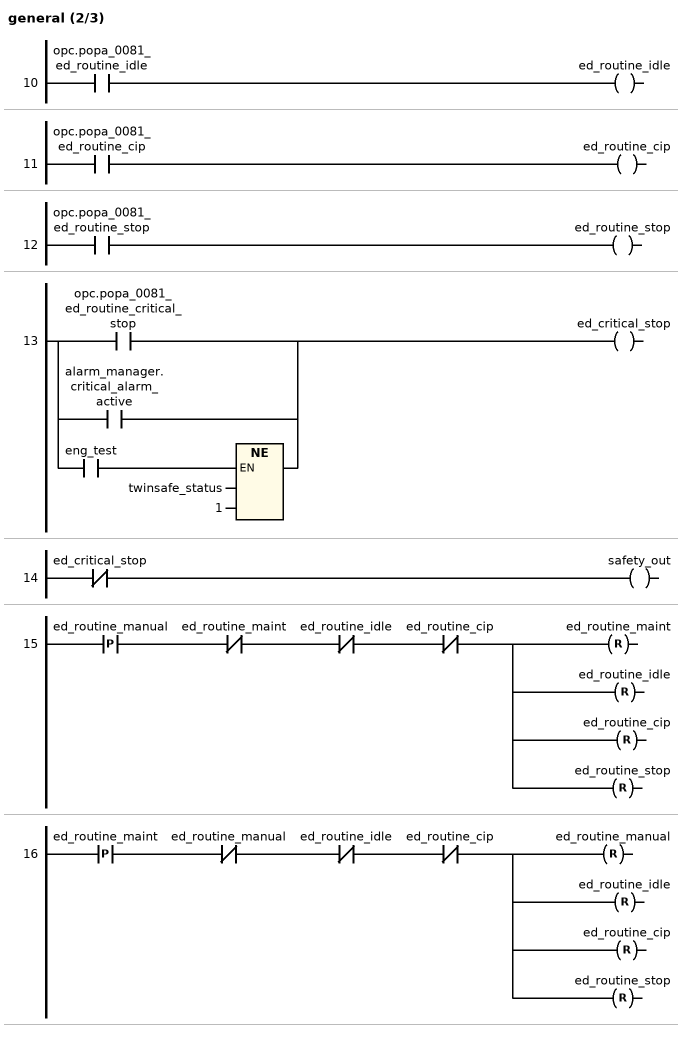
// NETWORK 10
ed_routine_idle := opc.popa_0081_ed_routine_idle;

// NETWORK 11
ed_routine_cip := opc.popa_0081_ed_routine_cip;

// NETWORK 12
ed_routine_stop := opc.popa_0081_ed_routine_stop;

// NETWORK 13
ed_critical_stop := opc.popa_0081_ed_routine_critical_stop OR alarm_manager.critical_alarm_active OR eng_test AND twinsafe_status <> 1;

// NETWORK 14
safety_out := NOT ed_critical_stop;

// NETWORK 15
_rt1(CLK := ed_routine_manual);
_w1 := _rt1.Q AND NOT ed_routine_maint AND NOT ed_routine_idle AND NOT ed_routine_cip;
ed_routine_maint R= _w1;
ed_routine_idle R= _w1;
ed_routine_cip R= _w1;
ed_routine_stop R= _w1;

// NETWORK 16
_rt2(CLK := ed_routine_maint);
_w2 := _rt2.Q AND NOT ed_routine_manual AND NOT ed_routine_idle AND NOT ed_routine_cip;
ed_routine_manual R= _w2;
ed_routine_idle R= _w2;
ed_routine_cip R= _w2;
ed_routine_stop R= _w2;

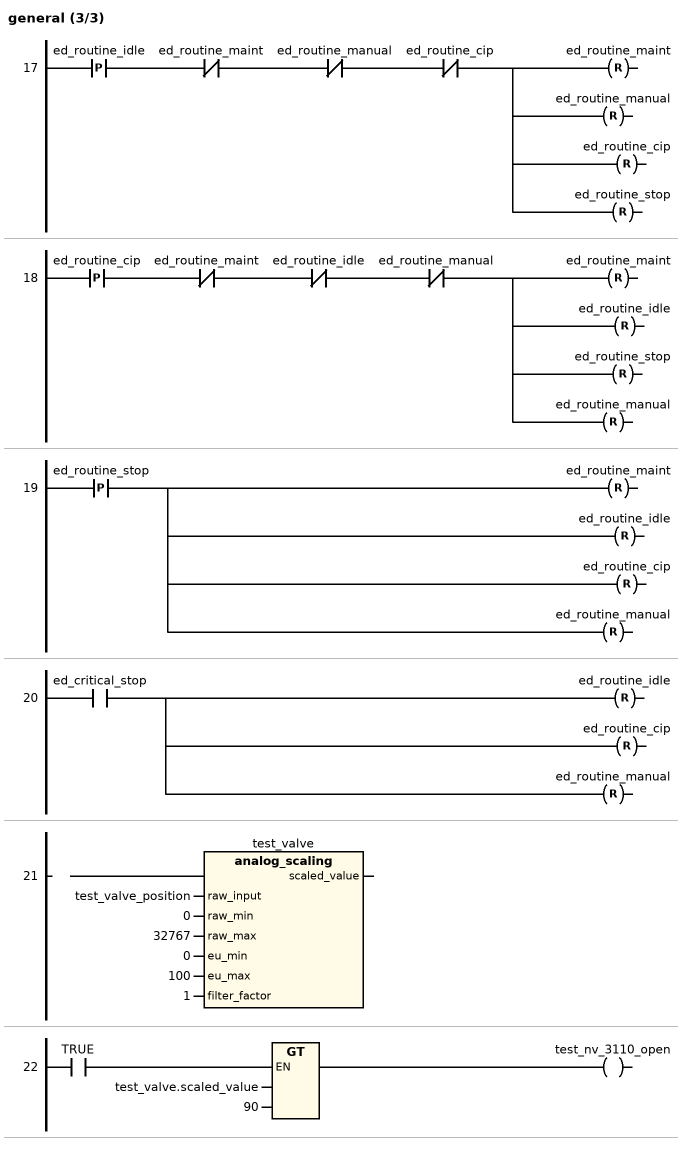
// NETWORK 17
_rt3(CLK := ed_routine_idle);
_w3 := _rt3.Q AND NOT ed_routine_maint AND NOT ed_routine_manual AND NOT ed_routine_cip;
ed_routine_maint R= _w3;
ed_routine_manual R= _w3;
ed_routine_cip R= _w3;
ed_routine_stop R= _w3;

// NETWORK 18
_rt4(CLK := ed_routine_cip);
_w4 := _rt4.Q AND NOT ed_routine_maint AND NOT ed_routine_idle AND NOT ed_routine_manual;
ed_routine_maint R= _w4;
ed_routine_idle R= _w4;
ed_routine_stop R= _w4;
ed_routine_manual R= _w4;

// NETWORK 19
_rt5(CLK := ed_routine_stop);
ed_routine_maint R= _rt5.Q;
ed_routine_idle R= _rt5.Q;
ed_routine_cip R= _rt5.Q;
ed_routine_manual R= _rt5.Q;

// NETWORK 20
ed_routine_idle R= ed_critical_stop;
ed_routine_cip R= ed_critical_stop;
ed_routine_manual R= ed_critical_stop;

// NETWORK 21
test_valve(
    raw_input := test_valve_position,
    raw_min := 0,
    raw_max := 32767,
    eu_min := 0,
    eu_max := 100,
    filter_factor := 1); // analog_scaling

// NETWORK 22
test_nv_3110_open := test_valve.scaled_value > 90;

END_PROGRAM

// ---- POUs/alarm_manager.TcPOU
PROGRAM alarm_manager
VAR
	critical_alarm_active: BOOL;
	error_alarm_active: BOOL;
	warning_alarm_active: BOOL;
	safety_status AT %I*: BOOL;
END_VAR

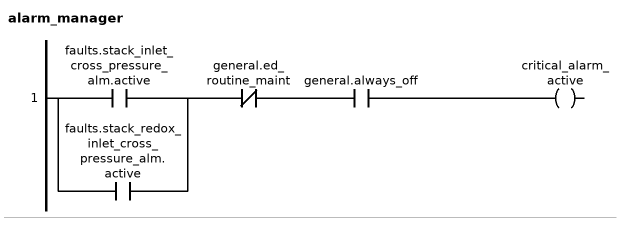
// NETWORK 1
critical_alarm_active := (faults.stack_inlet_cross_pressure_alm.active OR faults.stack_redox_inlet_cross_pressure_alm.active) AND NOT general.ed_routine_maint AND general.always_off;

END_PROGRAM

// ---- POUs/faults.TcPOU
PROGRAM faults
VAR PERSISTENT

//---Equipment Failure Faults----------------------------------------------------------------------------------------------

	//Discrete alarm example.  Replace with your own alarms
	u_3112_a_fail_to_start : alarm;
	u_3212_a_fail_to_start : alarm;
	u_3312_a_fail_to_start : alarm;
	u_3160_a_fail_to_start : alarm;
	u_3260_a_fail_to_start : alarm;
	u_3360_a_fail_to_start : alarm;
	u_3370_a_fail_to_start : alarm;
	u_3405_a_fail_to_start : alarm;
	// Discrete Alarm Example
	u_3112_a_fail_to_stop: Alarm;
	u_3212_a_fail_to_stop: Alarm;
	u_3312_a_fail_to_stop: Alarm;
	u_3160_a_fail_to_stop: Alarm;
	u_3260_a_fail_to_stop: Alarm;
	u_3360_a_fail_to_stop: Alarm;
	u_3370_a_fail_to_stop: Alarm;
	u_3405_a_fail_to_stop: Alarm;

	// Example analog valve position fail alarm
	av_3148_a_position_fail: Alarm;
	av_3248_a_position_fail: Alarm;
	av_3348_a_position_fail: Alarm;
	// Example digital valve fail to open alarm
	nv_3110_a_fail_to_open: Alarm;
	nv_3210_a_fail_to_open: Alarm;
	nv_3310_a_fail_to_open: Alarm;
	nv_3135_a_fail_to_open: Alarm;
	nv_3235_a_fail_to_open: Alarm;
	nv_3335_a_fail_to_open: Alarm;
	nv_3372_a_fail_to_open: Alarm;
	nv_3162_a_fail_to_open: Alarm;
	// Example digital valve fail to close alarm
	nv_3110_a_fail_to_close: Alarm;
	nv_3210_a_fail_to_close: Alarm;
	nv_3310_a_fail_to_close: Alarm;
	nv_3135_a_fail_to_close: Alarm;
	nv_3235_a_fail_to_close: Alarm;
	nv_3335_a_fail_to_close: Alarm;
	nv_3372_a_fail_to_close: Alarm;
	nv_3162_a_fail_to_close: Alarm;
	


//---Sensor threshold alarms----------------------------------------
	// Analog alarm low low
	cct_3120_a_low_low: Alarm;
	cct_3142_a_low_low: Alarm;
	cct_3220_a_low_low: Alarm;
	cct_3242_a_low_low: Alarm;
	cct_3320_a_low_low: Alarm;
	cct_3342_a_low_low: Alarm;
	cct_3413_a_low_low: Alarm;
	cgt_3910_a_low_low: Alarm;
	cpt_3144_a_low_low: Alarm;
	cpt_3158_a_low_low: Alarm;
	cpt_3407_a_low_low: Alarm;
	et_3711_a_low_low: Alarm;
	ft_3122_a_low_low: Alarm;
	ft_3222_a_low_low: Alarm;
	ft_3322_a_low_low: Alarm;
	it_3702_a_low_low: Alarm;
	lit_3905_a_low_low: Alarm;
	lit_3906_a_low_low: Alarm;
	lit_3907_a_low_low: Alarm;
	lit_3908_a_low_low: Alarm;
	lit_3915_a_low_low: Alarm;
	lt_3102_a_low_low: Alarm;
	lt_3153_a_low_low: Alarm;
	lt_3202_a_low_low: Alarm;
	lt_3253_a_low_low: Alarm;
	lt_3302_a_low_low: Alarm;
	lt_3353_a_low_low: Alarm;
	lt_3402_a_low_low: Alarm;
	pt_3119_a_low_low: Alarm;
	pt_3141_a_low_low: Alarm;
	pt_3219_a_low_low: Alarm;
	pt_3241_a_low_low: Alarm;
	pt_3319_a_low_low: Alarm;
	pt_3341_a_low_low: Alarm;
	pt_3414_a_low_low: Alarm;
	pt_3428_a_low_low: Alarm;
	tt_3118_a_low_low: Alarm;
	tt_3140_a_low_low: Alarm;
	tt_3218_a_low_low: Alarm;
	tt_3240_a_low_low: Alarm;
	tt_3318_a_low_low: Alarm;
	tt_3340_a_low_low: Alarm;
	tt_3432_a_low_low: Alarm;
	tt_3601_a_low_low: Alarm;


	// Analog alarm low
	cct_3120_a_low: Alarm;
	cct_3142_a_low: Alarm;
	cct_3220_a_low: Alarm;
	cct_3242_a_low: Alarm;
	cct_3320_a_low: Alarm;
	cct_3342_a_low: Alarm;
	cct_3413_a_low: Alarm;
	cgt_3910_a_low: Alarm;
	cpt_3144_a_low: Alarm;
	cpt_3158_a_low: Alarm;
	cpt_3407_a_low: Alarm;
	et_3711_a_low: Alarm;
	ft_3122_a_low: Alarm;
	ft_3222_a_low: Alarm;
	ft_3322_a_low: Alarm;
	it_3702_a_low: Alarm;
	lit_3905_a_low: Alarm;
	lit_3906_a_low: Alarm;
	lit_3907_a_low: Alarm;
	lit_3908_a_low: Alarm;
	lit_3915_a_low: Alarm;
	lt_3102_a_low: Alarm;
	lt_3153_a_low: Alarm;
	lt_3202_a_low: Alarm;
	lt_3253_a_low: Alarm;
	lt_3302_a_low: Alarm;
	lt_3353_a_low: Alarm;
	lt_3402_a_low: Alarm;
	pt_3119_a_low: Alarm;
	pt_3141_a_low: Alarm;
	pt_3219_a_low: Alarm;
	pt_3241_a_low: Alarm;
	pt_3319_a_low: Alarm;
	pt_3341_a_low: Alarm;
	pt_3414_a_low: Alarm;
	pt_3428_a_low: Alarm;
	tt_3118_a_low: Alarm;
	tt_3140_a_low: Alarm;
	tt_3218_a_low: Alarm;
	tt_3240_a_low: Alarm;
	tt_3318_a_low: Alarm;
	tt_3340_a_low: Alarm;
	tt_3432_a_low: Alarm;
	tt_3601_a_low: Alarm;


	// Analog alarm high
		cct_3120_a_high: Alarm;
	cct_3142_a_high: Alarm;
	cct_3220_a_high: Alarm;
	cct_3242_a_high: Alarm;
	cct_3320_a_high: Alarm;
	cct_3342_a_high: Alarm;
	cct_3413_a_high: Alarm;
	cgt_3910_a_high: Alarm;
	cpt_3144_a_high: Alarm;
	cpt_3158_a_high: Alarm;
	cpt_3407_a_high: Alarm;
	et_3711_a_high: Alarm;
	ft_3122_a_high: Alarm;
	ft_3222_a_high: Alarm;
	ft_3322_a_high: Alarm;
	it_3702_a_high: Alarm;
	lit_3905_a_high: Alarm;
	lit_3906_a_high: Alarm;
	lit_3907_a_high: Alarm;
	lit_3908_a_high: Alarm;
	lit_3915_a_high: Alarm;
	lt_3102_a_high: Alarm;
	lt_3153_a_high: Alarm;
	lt_3202_a_high: Alarm;
	lt_3253_a_high: Alarm;
	lt_3302_a_high: Alarm;
	lt_3353_a_high: Alarm;
	lt_3402_a_high: Alarm;
	pt_3119_a_high: Alarm;
	pt_3141_a_high: Alarm;
	pt_3219_a_high: Alarm;
	pt_3241_a_high: Alarm;
	pt_3319_a_high: Alarm;
	pt_3341_a_high: Alarm;
	pt_3414_a_high: Alarm;
	pt_3428_a_high: Alarm;
	tt_3118_a_high: Alarm;
	tt_3140_a_high: Alarm;
	tt_3218_a_high: Alarm;
	tt_3240_a_high: Alarm;
	tt_3318_a_high: Alarm;
	tt_3340_a_high: Alarm;
	tt_3432_a_high: Alarm;
	tt_3601_a_high: Alarm;


	// Analog alarm high high
		cct_3120_a_high_high: Alarm;
	cct_3142_a_high_high: Alarm;
	cct_3220_a_high_high: Alarm;
	cct_3242_a_high_high: Alarm;
	cct_3320_a_high_high: Alarm;
	cct_3342_a_high_high: Alarm;
	cct_3413_a_high_high: Alarm;
	cgt_3910_a_high_high: Alarm;
	cpt_3144_a_high_high: Alarm;
	cpt_3158_a_high_high: Alarm;
	cpt_3407_a_high_high: Alarm;
	et_3711_a_high_high: Alarm;
	ft_3122_a_high_high: Alarm;
	ft_3222_a_high_high: Alarm;
	ft_3322_a_high_high: Alarm;
	it_3702_a_high_high: Alarm;
	lit_3905_a_high_high: Alarm;
	lit_3906_a_high_high: Alarm;
	lit_3907_a_high_high: Alarm;
	lit_3908_a_high_high: Alarm;
	lit_3915_a_high_high: Alarm;
	lt_3102_a_high_high: Alarm;
	lt_3153_a_high_high: Alarm;
	lt_3202_a_high_high: Alarm;
	lt_3253_a_high_high: Alarm;
	lt_3302_a_high_high: Alarm;
	lt_3353_a_high_high: Alarm;
	lt_3402_a_high_high: Alarm;
	pt_3119_a_high_high: Alarm;
	pt_3141_a_high_high: Alarm;
	pt_3219_a_high_high: Alarm;
	pt_3241_a_high_high: Alarm;
	pt_3319_a_high_high: Alarm;
	pt_3341_a_high_high: Alarm;
	pt_3414_a_high_high: Alarm;
	pt_3428_a_high_high: Alarm;
	tt_3118_a_high_high: Alarm;
	tt_3140_a_high_high: Alarm;
	tt_3218_a_high_high: Alarm;
	tt_3240_a_high_high: Alarm;
	tt_3318_a_high_high: Alarm;
	tt_3340_a_high_high: Alarm;
	tt_3432_a_high_high: Alarm;
	tt_3601_a_high_high: Alarm;

//---System threshold alarms------------------------------------------------------------------------------------------------
	stack_inlet_cross_pressure_alm: Alarm;
	stack_redox_inlet_cross_pressure_alm: Alarm;
END_VAR
VAR
	salt_cross_pressure : REAL;
	acid_cross_pressure : REAL;
	base_cross_pressure : REAL;
	cross_pressure_cmp : REAL;
	redox_cross_pressure_cmp : REAL;
	max_inlet_pressure : REAL;
	min_inlet_pressure : REAL;
END_VAR

//Instantiate the alarm block, and map the inputs from the OPC GVL
(*u_3160_a_fail_to_start();
u_3160_a_fail_to_start.alm_ack:=opc.popa_0081_alarm_ack;
u_3160_a_fail_to_start.reset:=opc.popa_0081_alarm_reset;
u_3160_a_fail_to_start.priority:=opc.popa_0081_u_3160_a_fail_to_start_priority;
u_3160_a_fail_to_start.delay_setpoint:=opc.popa_0081_u_3160_a_fail_to_start_delay_setpoint;
u_3160_a_fail_to_start.enable:=opc.popa_0081_u_3160_a_fail_to_start_enable;

//Place your alarm trigger logic here.  
(*IF motor_starter_control.u_3160_a.run_command=TRUE AND motor_starter_control.u_3160_a.run_feedback=FALSE THEN
	u_3160_a_fail_to_start.trigger:=TRUE;
	ELSE
		u_3160_a_fail_to_start.trigger:=False;
	END_IF
	*)
//Instantiate the alarm block, and map the inputs from the OPC GVL
u_3160_a_fail_to_stop();
u_3160_a_fail_to_stop.alm_ack:=opc.popa_0081_alarm_ack;
u_3160_a_fail_to_stop.reset:=opc.popa_0081_alarm_reset;
u_3160_a_fail_to_stop.priority:=opc.popa_0081_u_3160_a_fail_to_stop_priority;
u_3160_a_fail_to_stop.delay_setpoint:=opc.popa_0081_u_3160_a_fail_to_stop_delay_setpoint;
u_3160_a_fail_to_stop.enable:=opc.popa_0081_u_3160_a_fail_to_stop_enable;

//Place your alarm trigger logic here.  
(*IF motor_starter_control.u_3160_a.run_command=FALSE AND motor_starter_control.u_3160_a.run_feedback=TRUE THEN
	u_3160_a_fail_to_stop.trigger:=TRUE;
	ELSE
		u_3160_a_fail_to_stop.trigger:=FALSE;
	END_IF
*)	*)

//---Pumps------------------------------------------------------------------------------------------------------------------------------------
//u_3112----------------------------------------------------------------------------------------------------------------
//Instantiate the alarm block, and map the inputs from the OPC GVL
u_3112_a_fail_to_start();
u_3112_a_fail_to_start.alm_ack:=opc.popa_0081_alarm_ack;
u_3112_a_fail_to_start.reset:=opc.popa_0081_alarm_reset;
u_3112_a_fail_to_start.priority:=opc.popa_0081_u_3112_a_fail_to_start_priority;
u_3112_a_fail_to_start.delay_setpoint:=opc.popa_0081_u_3112_a_fail_to_start_delay_setpoint;
u_3112_a_fail_to_start.enable:=opc.popa_0081_u_3112_a_fail_to_start_enable;

//Place your alarm trigger logic here.  
IF pump_manager.u_3112_a.run_command = TRUE AND pump_manager.u_3112_a.run_feedback=FALSE THEN
	u_3112_a_fail_to_start.trigger:=TRUE;
	ELSE
		u_3112_a_fail_to_start.trigger:=FALSE;
	END_IF
	
//Instantiate the alarm block, and map the inputs from the OPC GVL
u_3112_a_fail_to_stop();
u_3112_a_fail_to_stop.alm_ack:=opc.popa_0081_alarm_ack;
u_3112_a_fail_to_stop.reset:=opc.popa_0081_alarm_reset;
u_3112_a_fail_to_stop.priority:=opc.popa_0081_u_3112_a_fail_to_stop_priority;
u_3112_a_fail_to_stop.delay_setpoint:=opc.popa_0081_u_3112_a_fail_to_stop_delay_setpoint;
u_3112_a_fail_to_stop.enable:=opc.popa_0081_u_3112_a_fail_to_stop_enable;

//Place your alarm trigger logic here.  
IF pump_manager.u_3112_a.run_command = FALSE AND pump_manager.u_3112_a.run_feedback=TRUE THEN
	u_3112_a_fail_to_stop.trigger:=TRUE;
	ELSE
		u_3112_a_fail_to_stop.trigger:=FALSE;
	END_IF

//u_3212----------------------------------------------------------------------------------------------------------------
//Instantiate the alarm block, and map the inputs from the OPC GVL
u_3212_a_fail_to_start();
u_3212_a_fail_to_start.alm_ack:=opc.popa_0081_alarm_ack;
u_3212_a_fail_to_start.reset:=opc.popa_0081_alarm_reset;
u_3212_a_fail_to_start.priority:=opc.popa_0081_u_3212_a_fail_to_start_priority;
u_3212_a_fail_to_start.delay_setpoint:=opc.popa_0081_u_3212_a_fail_to_start_delay_setpoint;
u_3212_a_fail_to_start.enable:=opc.popa_0081_u_3212_a_fail_to_start_enable;

//Place your alarm trigger logic here.  
IF pump_manager.u_3212_a.run_command = TRUE AND pump_manager.u_3212_a.run_feedback=FALSE THEN
	u_3212_a_fail_to_start.trigger:=TRUE;
	ELSE
		u_3212_a_fail_to_start.trigger:=FALSE;
	END_IF
	
//Instantiate the alarm block, and map the inputs from the OPC GVL
u_3212_a_fail_to_stop();
u_3212_a_fail_to_stop.alm_ack:=opc.popa_0081_alarm_ack;
u_3212_a_fail_to_stop.reset:=opc.popa_0081_alarm_reset;
u_3212_a_fail_to_stop.priority:=opc.popa_0081_u_3212_a_fail_to_stop_priority;
u_3212_a_fail_to_stop.delay_setpoint:=opc.popa_0081_u_3212_a_fail_to_stop_delay_setpoint;
u_3212_a_fail_to_stop.enable:=opc.popa_0081_u_3212_a_fail_to_stop_enable;

//Place your alarm trigger logic here.  
IF pump_manager.u_3212_a.run_command = FALSE AND pump_manager.u_3212_a.run_feedback=TRUE THEN
	u_3212_a_fail_to_stop.trigger:=TRUE;
	ELSE
		u_3212_a_fail_to_stop.trigger:=FALSE;
	END_IF
	
//u_3312----------------------------------------------------------------------------------------------------------------
//Instantiate the alarm block, and map the inputs from the OPC GVL
u_3312_a_fail_to_start();
u_3312_a_fail_to_start.alm_ack:=opc.popa_0081_alarm_ack;
u_3312_a_fail_to_start.reset:=opc.popa_0081_alarm_reset;
u_3312_a_fail_to_start.priority:=opc.popa_0081_u_3312_a_fail_to_start_priority;
u_3312_a_fail_to_start.delay_setpoint:=opc.popa_0081_u_3312_a_fail_to_start_delay_setpoint;
u_3312_a_fail_to_start.enable:=opc.popa_0081_u_3312_a_fail_to_start_enable;

//Place your alarm trigger logic here.  
IF pump_manager.u_3312_a.run_command = TRUE AND pump_manager.u_3312_a.run_feedback=FALSE THEN
	u_3312_a_fail_to_start.trigger:=TRUE;
	ELSE
		u_3312_a_fail_to_start.trigger:=FALSE;
	END_IF
	
//Instantiate the alarm block, and map the inputs from the OPC GVL
u_3312_a_fail_to_stop();
u_3312_a_fail_to_stop.alm_ack:=opc.popa_0081_alarm_ack;
u_3312_a_fail_to_stop.reset:=opc.popa_0081_alarm_reset;
u_3312_a_fail_to_stop.priority:=opc.popa_0081_u_3312_a_fail_to_stop_priority;
u_3312_a_fail_to_stop.delay_setpoint:=opc.popa_0081_u_3312_a_fail_to_stop_delay_setpoint;
u_3312_a_fail_to_stop.enable:=opc.popa_0081_u_3312_a_fail_to_stop_enable;

//Place your alarm trigger logic here.  
IF pump_manager.u_3312_a.run_command = FALSE AND pump_manager.u_3312_a.run_feedback=TRUE THEN
	u_3312_a_fail_to_stop.trigger:=TRUE;
	ELSE
		u_3312_a_fail_to_stop.trigger:=FALSE;
	END_IF
	
//u_3405----------------------------------------------------------------------------------------------------------------
//Instantiate the alarm block, and map the inputs from the OPC GVL
u_3405_a_fail_to_start();
u_3405_a_fail_to_start.alm_ack:=opc.popa_0081_alarm_ack;
u_3405_a_fail_to_start.reset:=opc.popa_0081_alarm_reset;
//u_3405_a_fail_to_start.priority:=opc.popa_0081_u_3405_a_fail_to_start_priority;
//u_3405_a_fail_to_start.delay_setpoint:=opc.popa_0081_u_3405_a_fail_to_start_delay_setpoint;
//u_3405_a_fail_to_start.enable:=opc.popa_0081_u_3405_a_fail_to_start_enable;

//Place your alarm trigger logic here.  
IF pump_manager.u_3405_a.run_command = TRUE AND pump_manager.u_3405_a.run_feedback=FALSE THEN
	u_3405_a_fail_to_start.trigger:=TRUE;
	ELSE
		u_3405_a_fail_to_start.trigger:=FALSE;
	END_IF
	
//Instantiate the alarm block, and map the inputs from the OPC GVL
u_3405_a_fail_to_stop();
u_3405_a_fail_to_stop.alm_ack:=opc.popa_0081_alarm_ack;
u_3405_a_fail_to_stop.reset:=opc.popa_0081_alarm_reset;
//u_3405_a_fail_to_stop.priority:=opc.popa_0081_u_3405_a_fail_to_stop_priority;
//u_3405_a_fail_to_stop.delay_setpoint:=opc.popa_0081_u_3405_a_fail_to_stop_delay_setpoint;
//u_3405_a_fail_to_stop.enable:=opc.popa_0081_u_3405_a_fail_to_stop_enable;

//Place your alarm trigger logic here.  
IF pump_manager.u_3405_a.run_command = FALSE AND pump_manager.u_3405_a.run_feedback=TRUE THEN
	u_3405_a_fail_to_stop.trigger:=TRUE;
	ELSE
		u_3405_a_fail_to_stop.trigger:=FALSE;
	END_IF

//u_3160----------------------------------------------------------------------------------------------------------------
//Instantiate the alarm block, and map the inputs from the OPC GVL
u_3160_a_fail_to_start();
u_3160_a_fail_to_start.alm_ack:=opc.popa_0081_alarm_ack;
u_3160_a_fail_to_start.reset:=opc.popa_0081_alarm_reset;
u_3160_a_fail_to_start.priority:=opc.popa_0081_u_3160_a_fail_to_start_priority;
u_3160_a_fail_to_start.delay_setpoint:=opc.popa_0081_u_3160_a_fail_to_start_delay_setpoint;
u_3160_a_fail_to_start.enable:=opc.popa_0081_u_3160_a_fail_to_start_enable;

//Place your alarm trigger logic here.  
IF pump_manager.u_3160_a.run_command = TRUE AND pump_manager.u_3160_a.run_feedback=FALSE THEN
	u_3160_a_fail_to_start.trigger:=TRUE;
	ELSE
		u_3160_a_fail_to_start.trigger:=FALSE;
	END_IF
	
//Instantiate the alarm block, and map the inputs from the OPC GVL
u_3160_a_fail_to_stop();
u_3160_a_fail_to_stop.alm_ack:=opc.popa_0081_alarm_ack;
u_3160_a_fail_to_stop.reset:=opc.popa_0081_alarm_reset;
u_3160_a_fail_to_stop.priority:=opc.popa_0081_u_3160_a_fail_to_stop_priority;
u_3160_a_fail_to_stop.delay_setpoint:=opc.popa_0081_u_3160_a_fail_to_stop_delay_setpoint;
u_3160_a_fail_to_stop.enable:=opc.popa_0081_u_3160_a_fail_to_stop_enable;

//Place your alarm trigger logic here.  
IF pump_manager.u_3160_a.run_command = FALSE AND pump_manager.u_3160_a.run_feedback=TRUE THEN
	u_3160_a_fail_to_stop.trigger:=TRUE;
	ELSE
		u_3160_a_fail_to_stop.trigger:=FALSE;
	END_IF
	
	
//u_3260----------------------------------------------------------------------------------------------------------------
//Instantiate the alarm block, and map the inputs from the OPC GVL
u_3260_a_fail_to_start();
u_3260_a_fail_to_start.alm_ack:=opc.popa_0081_alarm_ack;
u_3260_a_fail_to_start.reset:=opc.popa_0081_alarm_reset;
u_3260_a_fail_to_start.priority:=opc.popa_0081_u_3260_a_fail_to_start_priority;
u_3260_a_fail_to_start.delay_setpoint:=opc.popa_0081_u_3260_a_fail_to_start_delay_setpoint;
u_3260_a_fail_to_start.enable:=opc.popa_0081_u_3260_a_fail_to_start_enable;

//Place your alarm trigger logic here.  
IF pump_manager.u_3260_a.run_command = TRUE AND pump_manager.u_3260_a.run_feedback=FALSE THEN
	u_3260_a_fail_to_start.trigger:=TRUE;
	ELSE
		u_3260_a_fail_to_start.trigger:=FALSE;
	END_IF
	
//Instantiate the alarm block, and map the inputs from the OPC GVL
u_3260_a_fail_to_stop();
u_3260_a_fail_to_stop.alm_ack:=opc.popa_0081_alarm_ack;
u_3260_a_fail_to_stop.reset:=opc.popa_0081_alarm_reset;
u_3260_a_fail_to_stop.priority:=opc.popa_0081_u_3260_a_fail_to_stop_priority;
u_3260_a_fail_to_stop.delay_setpoint:=opc.popa_0081_u_3260_a_fail_to_stop_delay_setpoint;
u_3260_a_fail_to_stop.enable:=opc.popa_0081_u_3260_a_fail_to_stop_enable;

//Place your alarm trigger logic here.  
IF pump_manager.u_3260_a.run_command = FALSE AND pump_manager.u_3260_a.run_feedback=TRUE THEN
	u_3260_a_fail_to_stop.trigger:=TRUE;
	ELSE
		u_3260_a_fail_to_stop.trigger:=FALSE;
	END_IF
	
//u_3360----------------------------------------------------------------------------------------------------------------
//Instantiate the alarm block, and map the inputs from the OPC GVL
u_3360_a_fail_to_start();
u_3360_a_fail_to_start.alm_ack:=opc.popa_0081_alarm_ack;
u_3360_a_fail_to_start.reset:=opc.popa_0081_alarm_reset;
u_3360_a_fail_to_start.priority:=opc.popa_0081_u_3360_a_fail_to_start_priority;
u_3360_a_fail_to_start.delay_setpoint:=opc.popa_0081_u_3360_a_fail_to_start_delay_setpoint;
u_3360_a_fail_to_start.enable:=opc.popa_0081_u_3360_a_fail_to_start_enable;

//Place your alarm trigger logic here.  
IF pump_manager.u_3360_a.run_command = TRUE AND pump_manager.u_3360_a.run_feedback=FALSE THEN
	u_3360_a_fail_to_start.trigger:=TRUE;
	ELSE
		u_3360_a_fail_to_start.trigger:=FALSE;
	END_IF
	
//Instantiate the alarm block, and map the inputs from the OPC GVL
u_3360_a_fail_to_stop();
u_3360_a_fail_to_stop.alm_ack:=opc.popa_0081_alarm_ack;
u_3360_a_fail_to_stop.reset:=opc.popa_0081_alarm_reset;
u_3360_a_fail_to_stop.priority:=opc.popa_0081_u_3360_a_fail_to_stop_priority;
u_3360_a_fail_to_stop.delay_setpoint:=opc.popa_0081_u_3360_a_fail_to_stop_delay_setpoint;
u_3360_a_fail_to_stop.enable:=opc.popa_0081_u_3360_a_fail_to_stop_enable;

//Place your alarm trigger logic here.  
IF pump_manager.u_3360_a.run_command = FALSE AND pump_manager.u_3360_a.run_feedback=TRUE THEN
	u_3360_a_fail_to_stop.trigger:=TRUE;
	ELSE
		u_3360_a_fail_to_stop.trigger:=FALSE;
	END_IF
	
//u_3370----------------------------------------------------------------------------------------------------------------
//Instantiate the alarm block, and map the inputs from the OPC GVL
u_3370_a_fail_to_start();
u_3370_a_fail_to_start.alm_ack:=opc.popa_0081_alarm_ack;
u_3370_a_fail_to_start.reset:=opc.popa_0081_alarm_reset;
u_3370_a_fail_to_start.priority:=opc.popa_0081_u_3370_a_fail_to_start_priority;
u_3370_a_fail_to_start.delay_setpoint:=opc.popa_0081_u_3370_a_fail_to_start_delay_setpoint;
u_3370_a_fail_to_start.enable:=opc.popa_0081_u_3370_a_fail_to_start_enable;

//Place your alarm trigger logic here.  
IF pump_manager.u_3370_a.run_command = TRUE AND pump_manager.u_3370_a.run_feedback=FALSE THEN
	u_3370_a_fail_to_start.trigger:=TRUE;
	ELSE
		u_3370_a_fail_to_start.trigger:=FALSE;
	END_IF
	
//Instantiate the alarm block, and map the inputs from the OPC GVL
u_3370_a_fail_to_stop();
u_3370_a_fail_to_stop.alm_ack:=opc.popa_0081_alarm_ack;
u_3370_a_fail_to_stop.reset:=opc.popa_0081_alarm_reset;
u_3370_a_fail_to_stop.priority:=opc.popa_0081_u_3370_a_fail_to_stop_priority;
u_3370_a_fail_to_stop.delay_setpoint:=opc.popa_0081_u_3370_a_fail_to_stop_delay_setpoint;
u_3370_a_fail_to_stop.enable:=opc.popa_0081_u_3370_a_fail_to_stop_enable;

//Place your alarm trigger logic here.  
IF pump_manager.u_3370_a.run_command = FALSE AND pump_manager.u_3370_a.run_feedback=TRUE THEN
	u_3370_a_fail_to_stop.trigger:=TRUE;
	ELSE
		u_3370_a_fail_to_stop.trigger:=FALSE;
	END_IF
	

//---Valves---------------------------------------------------------------------------------------------------------------------------------------------------------------
//Instantiate the alarm block, and map the inputs from the OPC GVL
av_3148_a_position_fail();
av_3148_a_position_fail.alm_ack:=opc.popa_0081_alarm_ack;
av_3148_a_position_fail.reset:=opc.popa_0081_alarm_reset;
av_3148_a_position_fail.priority:=opc.popa_0081_av_3148_a_position_fail_priority;
av_3148_a_position_fail.delay_setpoint:=opc.popa_0081_av_3148_a_position_fail_delay_setpoint;
av_3148_a_position_fail.enable:=opc.popa_0081_av_3148_a_position_fail_enable;

//Place your alarm trigger logic here.  
IF io_mapping.av_3148_a_position_feedback.scaled_value>valve_manager.av_3148_a.position_deadband_high OR io_mapping.av_3148_a_position_feedback.scaled_value<valve_manager.av_3148.position_deadband_low THEN
	av_3148_a_position_fail.trigger:=TRUE;
	ELSE
		av_3148_a_position_fail.trigger:=FALSE;
	END_IF
	
//Instantiate the alarm block, and map the inputs from the OPC GVL
nv_3372_a_fail_to_open();
nv_3372_a_fail_to_open.alm_ack:=opc.popa_0081_alarm_ack;
nv_3372_a_fail_to_open.reset:=opc.popa_0081_alarm_reset;
nv_3372_a_fail_to_open.priority:=opc.popa_0081_nv_3372_a_fail_to_open_priority;
nv_3372_a_fail_to_open.delay_setpoint:=opc.popa_0081_nv_3372_a_fail_to_open_delay_setpoint;
nv_3372_a_fail_to_open.enable:=opc.popa_0081_nv_3372_a_fail_to_open_enable;

//Place your alarm trigger logic here.  
IF valve_manager.nv_3372_a.open_command=TRUE AND valve_manager.nv_3372_a.open_feedback=FALSE THEN
	nv_3372_a_fail_to_open.trigger:=TRUE;
	ELSE
		nv_3372_a_fail_to_open.trigger:=FALSE;
	END_IF
	
//Instantiate the alarm block, and map the inputs from the OPC GVL
nv_3372_a_fail_to_close();
nv_3372_a_fail_to_close.alm_ack:=opc.popa_0081_alarm_ack;
nv_3372_a_fail_to_close.reset:=opc.popa_0081_alarm_reset;
nv_3372_a_fail_to_close.priority:=opc.popa_0081_nv_3372_a_fail_to_close_priority;
nv_3372_a_fail_to_close.delay_setpoint:=opc.popa_0081_nv_3372_a_fail_to_close_delay_setpoint;
nv_3372_a_fail_to_close.enable:=opc.popa_0081_nv_3372_a_fail_to_close_enable;

//Place your alarm trigger logic here.  
IF valve_manager.nv_3372_a.open_command=FALSE AND valve_manager.nv_3372_a.open_feedback=TRUE THEN
	nv_3372_a_fail_to_close.trigger:=TRUE;
	ELSE
		nv_3372_a_fail_to_close.trigger:=FALSE;
	END_IF	

	
//---System threshold alarms---------------------------------------------------------------------------------------------------

//Instantiate the alarm block, and map the inputs from the OPC GVL
stack_inlet_cross_pressure_alm();
stack_inlet_cross_pressure_alm.alm_ack:=opc.popa_0081_alarm_ack;
stack_inlet_cross_pressure_alm.reset:=opc.popa_0081_alarm_reset;
stack_inlet_cross_pressure_alm.priority:=3;//opc.popa_0081_nv_3372_a_fail_to_close_priority;
stack_inlet_cross_pressure_alm.delay_setpoint:= 1;//opc.popa_0081_nv_3372_a_fail_to_close_delay_setpoint;
stack_inlet_cross_pressure_alm.enable:=TRUE;//opc.popa_0081_nv_3372_a_fail_to_close_enable;

//Place your alarm trigger logic here.  
max_inlet_pressure := MAX(io_mapping.pt_3119_a.scaled_value, io_mapping.pt_3219_a.scaled_value, io_mapping.pt_3319_a.scaled_value); 
min_inlet_pressure := MIN(io_mapping.pt_3119_a.scaled_value, io_mapping.pt_3219_a.scaled_value, io_mapping.pt_3319_a.scaled_value);
cross_pressure_cmp :=(max_inlet_pressure - min_inlet_pressure); 
IF cross_pressure_cmp >= 0.1 THEN//OR (((io_mapping.pt_3119.scaled_value + io_mapping.pt_3141.scaled_value)/2) - io_mapping.pt_3414.scaled_value) >=0.1 THEN
	stack_inlet_cross_pressure_alm.trigger := TRUE;
	ELSE
		stack_inlet_cross_pressure_alm.trigger := FALSE;
END_IF

//Instantiate the alarm block, and map the inputs from the OPC GVL
stack_redox_inlet_cross_pressure_alm();
stack_redox_inlet_cross_pressure_alm.alm_ack:=opc.popa_0081_alarm_ack;
stack_redox_inlet_cross_pressure_alm.reset:=opc.popa_0081_alarm_reset;
stack_redox_inlet_cross_pressure_alm.priority:=3;//opc.popa_0081_nv_3372_a_fail_to_close_priority;
stack_redox_inlet_cross_pressure_alm.delay_setpoint:= 3;//opc.popa_0081_nv_3372_a_fail_to_close_delay_setpoint;
stack_redox_inlet_cross_pressure_alm.enable:=TRUE;//opc.popa_0081_nv_3372_a_fail_to_close_enable;

//Place your alarm trigger logic here.  
redox_cross_pressure_cmp :=ABS(((io_mapping.pt_3119_a.scaled_value + io_mapping.pt_3141_a.scaled_value)/2) - io_mapping.pt_3414_a.scaled_value);
IF  redox_cross_pressure_cmp >= 0.2 THEN
	stack_redox_inlet_cross_pressure_alm.trigger := TRUE;
	ELSE
		stack_redox_inlet_cross_pressure_alm.trigger := FALSE;
END_IF


//tt_3340-----------------------------------------------------------------------------------------------------
//Instantiate the alarm block, and map the inputs from the OPC GVL
tt_3340_a_high_high();
tt_3340_a_high_high.alm_ack:=opc.popa_0081_alarm_ack;
tt_3340_a_high_high.reset:=opc.popa_0081_alarm_reset;
tt_3340_a_high_high.priority:=opc.popa_0081_tt_3340_a_high_high_priority;
tt_3340_a_high_high.delay_setpoint:=opc.popa_0081_tt_3340_a_high_high_setpoint;
tt_3340_a_high_high.enable:=opc.popa_0081_tt_3340_a_high_high_enable;

//Timer delay elapsed
tt_3340_a_high_high.delay_ton_et;

//Place your alarm trigger logic here. 
IF io_mapping.tt_3340_a.scaled_value >= opc.popa_0081_tt_3340_a_high_high_setpoint THEN
    tt_3340_a_high_high.trigger := TRUE;
    ELSE
        tt_3340_a_high_high.trigger := FALSE;
END_IF

	
//cct_3120-----------------------------------------------------------------------------------------------------
//Instantiate the alarm block, and map the inputs from the OPC GVL
cct_3120_a_low();
cct_3120_a_low.alm_ack:=opc.popa_0081_alarm_ack;
cct_3120_a_low.reset:=opc.popa_0081_alarm_reset;
cct_3120_a_low.priority:=opc.popa_0081_cct_3120_a_low_priority;
cct_3120_a_low.delay_setpoint:=opc.popa_0081_cct_3120_a_low_setpoint;
cct_3120_a_low.enable:=opc.popa_0081_cct_3120_a_low_enable;

//Timer delay elapsed
cct_3120_a_low.delay_ton_et;

//Place your alarm trigger logic here. 
IF io_mapping.cct_3120_a.scaled_value < opc.popa_0081_cct_3120_a_low_setpoint THEN
    cct_3120_a_low.trigger := TRUE;
    ELSE
        cct_3120_a_low.trigger := FALSE;
END_IF
	
//cct_3120-----------------------------------------------------------------------------------------------------
//Instantiate the alarm block, and map the inputs from the OPC GVL
cct_3120_a_high();
cct_3120_a_high.alm_ack:=opc.popa_0081_alarm_ack;
cct_3120_a_high.reset:=opc.popa_0081_alarm_reset;
cct_3120_a_high.priority:=opc.popa_0081_cct_3120_a_high_priority;
cct_3120_a_high.delay_setpoint:=opc.popa_0081_cct_3120_a_high_setpoint;
cct_3120_a_high.enable:=opc.popa_0081_cct_3120_a_high_enable;

//Timer delay elapsed
cct_3120_a_high.delay_ton_et;

//Place your alarm trigger logic here. 
IF io_mapping.cct_3120_a.scaled_value > opc.popa_0081_cct_3120_a_high_setpoint THEN
    cct_3120_a_high.trigger := TRUE;
    ELSE
        cct_3120_a_high.trigger := FALSE;
END_IF
	
//cct_3120-----------------------------------------------------------------------------------------------------
//Instantiate the alarm block, and map the inputs from the OPC GVL
cct_3120_a_high_high();
cct_3120_a_high_high.alm_ack:=opc.popa_0081_alarm_ack;
cct_3120_a_high_high.reset:=opc.popa_0081_alarm_reset;
cct_3120_a_high_high.priority:=opc.popa_0081_cct_3120_a_high_high_priority;
cct_3120_a_high_high.delay_setpoint:=opc.popa_0081_cct_3120_a_high_high_setpoint;
cct_3120_a_high_high.enable:=opc.popa_0081_cct_3120_a_high_high_enable;

//Timer delay elapsed
cct_3120_a_high_high.delay_ton_et;

//Place your alarm trigger logic here. 
IF io_mapping.cct_3120_a.scaled_value >= opc.popa_0081_cct_3120_a_high_high_setpoint THEN
    cct_3120_a_high_high.trigger := TRUE;
    ELSE
        cct_3120_a_high_high.trigger := FALSE;
END_IF


//cct_3220-----------------------------------------------------------------------------------------------------
//Instantiate the alarm block, and map the inputs from the OPC GVL
cct_3220_a_low_low();
cct_3220_a_low_low.alm_ack:=opc.popa_0081_alarm_ack;
cct_3220_a_low_low.reset:=opc.popa_0081_alarm_reset;
cct_3220_a_low_low.priority:=opc.popa_0081_cct_3220_a_low_low_priority;
cct_3220_a_low_low.delay_setpoint:=opc.popa_0081_cct_3220_a_low_low_setpoint;
cct_3220_a_low_low.enable:=opc.popa_0081_cct_3220_a_low_low_enable;

//Timer delay elapsed
cct_3220_a_low_low.delay_ton_et;

//Place your alarm trigger logic here. 
IF io_mapping.cct_3220_a.scaled_value <= opc.popa_0081_cct_3220_a_low_low_setpoint THEN
    cct_3220_a_low_low.trigger := TRUE;
    ELSE
        cct_3220_a_low_low.trigger := FALSE;
END_IF
	
//cct_3220-----------------------------------------------------------------------------------------------------
//Instantiate the alarm block, and map the inputs from the OPC GVL
cct_3220_a_low();
cct_3220_a_low.alm_ack:=opc.popa_0081_alarm_ack;
cct_3220_a_low.reset:=opc.popa_0081_alarm_reset;
cct_3220_a_low.priority:=opc.popa_0081_cct_3220_a_low_priority;
cct_3220_a_low.delay_setpoint:=opc.popa_0081_cct_3220_a_low_setpoint;
cct_3220_a_low.enable:=opc.popa_0081_cct_3220_a_low_enable;

//Timer delay elapsed
cct_3220_a_low.delay_ton_et;

//Place your alarm trigger logic here. 
IF io_mapping.cct_3220_a.scaled_value < opc.popa_0081_cct_3220_a_low_setpoint THEN
    cct_3220_a_low.trigger := TRUE;
    ELSE
        cct_3220_a_low.trigger := FALSE;
END_IF
	
//cct_3220-----------------------------------------------------------------------------------------------------
//Instantiate the alarm block, and map the inputs from the OPC GVL
cct_3220_a_high();
cct_3220_a_high.alm_ack:=opc.popa_0081_alarm_ack;
cct_3220_a_high.reset:=opc.popa_0081_alarm_reset;
cct_3220_a_high.priority:=opc.popa_0081_cct_3220_a_high_priority;
cct_3220_a_high.delay_setpoint:=opc.popa_0081_cct_3220_a_high_setpoint;
cct_3220_a_high.enable:=opc.popa_0081_cct_3220_a_high_enable;

//Timer delay elapsed
cct_3220_a_high.delay_ton_et;

//Place your alarm trigger logic here. 
IF io_mapping.cct_3220_a.scaled_value > opc.popa_0081_cct_3220_a_high_setpoint THEN
    cct_3220_a_high.trigger := TRUE;
    ELSE
        cct_3220_a_high.trigger := FALSE;
END_IF
	
//cct_3220-----------------------------------------------------------------------------------------------------
//Instantiate the alarm block, and map the inputs from the OPC GVL
cct_3220_a_high_high();
cct_3220_a_high_high.alm_ack:=opc.popa_0081_alarm_ack;
cct_3220_a_high_high.reset:=opc.popa_0081_alarm_reset;
cct_3220_a_high_high.priority:=opc.popa_0081_cct_3220_a_high_high_priority;
cct_3220_a_high_high.delay_setpoint:=opc.popa_0081_cct_3220_a_high_high_setpoint;
cct_3220_a_high_high.enable:=opc.popa_0081_cct_3220_a_high_high_enable;

//Timer delay elapsed
cct_3220_a_high_high.delay_ton_et;

//Place your alarm trigger logic here. 
IF io_mapping.cct_3220_a.scaled_value >= opc.popa_0081_cct_3220_a_high_high_setpoint THEN
    cct_3220_a_high_high.trigger := TRUE;
    ELSE
        cct_3220_a_high_high.trigger := FALSE;
END_IF


//cct_3320-----------------------------------------------------------------------------------------------------
//Instantiate the alarm block, and map the inputs from the OPC GVL
cct_3320_a_low_low();
cct_3320_a_low_low.alm_ack:=opc.popa_0081_alarm_ack;
cct_3320_a_low_low.reset:=opc.popa_0081_alarm_reset;
cct_3320_a_low_low.priority:=opc.popa_0081_cct_3320_a_low_low_priority;
cct_3320_a_low_low.delay_setpoint:=opc.popa_0081_cct_3320_a_low_low_setpoint;
cct_3320_a_low_low.enable:=opc.popa_0081_cct_3320_a_low_low_enable;

//Timer delay elapsed
cct_3320_a_low_low.delay_ton_et;

//Place your alarm trigger logic here. 
IF io_mapping.cct_3320_a.scaled_value <= opc.popa_0081_cct_3320_a_low_low_setpoint THEN
    cct_3320_a_low_low.trigger := TRUE;
    ELSE
        cct_3320_a_low_low.trigger := FALSE;
END_IF
	
//cct_3320-----------------------------------------------------------------------------------------------------
//Instantiate the alarm block, and map the inputs from the OPC GVL
cct_3320_a_low();
cct_3320_a_low.alm_ack:=opc.popa_0081_alarm_ack;
cct_3320_a_low.reset:=opc.popa_0081_alarm_reset;
cct_3320_a_low.priority:=opc.popa_0081_cct_3320_a_low_priority;
cct_3320_a_low.delay_setpoint:=opc.popa_0081_cct_3320_a_low_setpoint;
cct_3320_a_low.enable:=opc.popa_0081_cct_3320_a_low_enable;

//Timer delay elapsed
cct_3320_a_low.delay_ton_et;

//Place your alarm trigger logic here. 
IF io_mapping.cct_3320_a.scaled_value < opc.popa_0081_cct_3320_a_low_setpoint THEN
    cct_3320_a_low.trigger := TRUE;
    ELSE
        cct_3320_a_low.trigger := FALSE;
END_IF
	
//cct_3320-----------------------------------------------------------------------------------------------------
//Instantiate the alarm block, and map the inputs from the OPC GVL
cct_3320_a_high();
cct_3320_a_high.alm_ack:=opc.popa_0081_alarm_ack;
cct_3320_a_high.reset:=opc.popa_0081_alarm_reset;
cct_3320_a_high.priority:=opc.popa_0081_cct_3320_a_high_priority;
cct_3320_a_high.delay_setpoint:=opc.popa_0081_cct_3320_a_high_setpoint;
cct_3320_a_high.enable:=opc.popa_0081_cct_3320_a_high_enable;

//Timer delay elapsed
cct_3320_a_high.delay_ton_et;

//Place your alarm trigger logic here. 
IF io_mapping.cct_3320_a.scaled_value > opc.popa_0081_cct_3320_a_high_setpoint THEN
    cct_3320_a_high.trigger := TRUE;
    ELSE
        cct_3320_a_high.trigger := FALSE;
END_IF
	
//cct_3320-----------------------------------------------------------------------------------------------------
//Instantiate the alarm block, and map the inputs from the OPC GVL
cct_3320_a_high_high();
cct_3320_a_high_high.alm_ack:=opc.popa_0081_alarm_ack;
cct_3320_a_high_high.reset:=opc.popa_0081_alarm_reset;
cct_3320_a_high_high.priority:=opc.popa_0081_cct_3320_a_high_high_priority;
cct_3320_a_high_high.delay_setpoint:=opc.popa_0081_cct_3320_a_high_high_setpoint;
cct_3320_a_high_high.enable:=opc.popa_0081_cct_3320_a_high_high_enable;

//Timer delay elapsed
cct_3320_a_high_high.delay_ton_et;

//Place your alarm trigger logic here. 
IF io_mapping.cct_3320_a.scaled_value >= opc.popa_0081_cct_3320_a_high_high_setpoint THEN
    cct_3320_a_high_high.trigger := TRUE;
    ELSE
        cct_3320_a_high_high.trigger := FALSE;
END_IF


//cct_3142-----------------------------------------------------------------------------------------------------
//Instantiate the alarm block, and map the inputs from the OPC GVL
cct_3142_a_low_low();
cct_3142_a_low_low.alm_ack:=opc.popa_0081_alarm_ack;
cct_3142_a_low_low.reset:=opc.popa_0081_alarm_reset;
cct_3142_a_low_low.priority:=opc.popa_0081_cct_3142_a_low_low_priority;
cct_3142_a_low_low.delay_setpoint:=opc.popa_0081_cct_3142_a_low_low_setpoint;
cct_3142_a_low_low.enable:=opc.popa_0081_cct_3142_a_low_low_enable;

//Timer delay elapsed
cct_3142_a_low_low.delay_ton_et;

//Place your alarm trigger logic here. 
IF io_mapping.cct_3142_a.scaled_value <= opc.popa_0081_cct_3142_a_low_low_setpoint THEN
    cct_3142_a_low_low.trigger := TRUE;
    ELSE
        cct_3142_a_low_low.trigger := FALSE;
END_IF
	
//cct_3142-----------------------------------------------------------------------------------------------------
//Instantiate the alarm block, and map the inputs from the OPC GVL
cct_3142_a_low();
cct_3142_a_low.alm_ack:=opc.popa_0081_alarm_ack;
cct_3142_a_low.reset:=opc.popa_0081_alarm_reset;
cct_3142_a_low.priority:=opc.popa_0081_cct_3142_a_low_priority;
cct_3142_a_low.delay_setpoint:=opc.popa_0081_cct_3142_a_low_setpoint;
cct_3142_a_low.enable:=opc.popa_0081_cct_3142_a_low_enable;

//Timer delay elapsed
cct_3142_a_low.delay_ton_et;

//Place your alarm trigger logic here. 
IF io_mapping.cct_3142_a.scaled_value < opc.popa_0081_cct_3142_a_low_setpoint THEN
    cct_3142_a_low.trigger := TRUE;
    ELSE
        cct_3142_a_low.trigger := FALSE;
END_IF
	
//cct_3142-----------------------------------------------------------------------------------------------------
//Instantiate the alarm block, and map the inputs from the OPC GVL
cct_3142_a_high();
cct_3142_a_high.alm_ack:=opc.popa_0081_alarm_ack;
cct_3142_a_high.reset:=opc.popa_0081_alarm_reset;
cct_3142_a_high.priority:=opc.popa_0081_cct_3142_a_high_priority;
cct_3142_a_high.delay_setpoint:=opc.popa_0081_cct_3142_a_high_setpoint;
cct_3142_a_high.enable:=opc.popa_0081_cct_3142_a_high_enable;

//Timer delay elapsed
cct_3142_a_high.delay_ton_et;

//Place your alarm trigger logic here. 
IF io_mapping.cct_3142_a.scaled_value > opc.popa_0081_cct_3142_a_high_setpoint THEN
    cct_3142_a_high.trigger := TRUE;
    ELSE
        cct_3142_a_high.trigger := FALSE;
END_IF
	
